{region " SIGNAL AREA : NAME->X_Pr_Axl3_Wh1 LENGTH->8 STARTBIT :0"}
Raw_X_Pr_Axl3_Wh1						:= _FB_CanRx_Message_224.X_Byte_0;
GVL.IIVD.X_Pr_Axl3_Wh1.e				:= (Raw_X_Pr_Axl3_Wh1 > 16#FD) AND (Raw_X_Pr_Axl3_Wh1 < 16#FF);
GVL.IIVD.X_Pr_Axl3_Wh1.na				:= (Raw_X_Pr_Axl3_Wh1 = 16#FF);
GVL.IIVD.X_Pr_Axl3_Wh1.RangeExcd		:= NOT ((USINT_TO_REAL(BYTE_TO_USINT(Raw_X_Pr_Axl3_Wh1)) >= 0) AND (USINT_TO_REAL(BYTE_TO_USINT(Raw_X_Pr_Axl3_Wh1)) <= 250));
GVL.IIVD.X_Pr_Axl3_Wh1.v				:= NOT( GVL.IIVD.S_TmOut_Lastik_Basinclari_2_0X224 OR GVL.IIVD.X_Pr_Axl3_Wh1.RangeExcd OR GVL.IIVD.X_Pr_Axl3_Wh1.e OR GVL.IIVD.X_Pr_Axl3_Wh1.na) ;
GVL.IIVD.X_Pr_Axl3_Wh1.x				:= 
(*SELECT 1 : Is data valid ?*)				SEL(GVL.IIVD.X_Pr_Axl3_Wh1.v,
(*DEFAULT value assigment*)					0,
(*Transmission is VALID*)					USINT_TO_REAL(BYTE_TO_USINT(Raw_X_Pr_Axl3_Wh1)));
{endregion}
{region " SIGNAL AREA : NAME->X_Pr_Axl3_Wh2 LENGTH->8 STARTBIT :8"}
Raw_X_Pr_Axl3_Wh2						:= _FB_CanRx_Message_224.X_Byte_1;
GVL.IIVD.X_Pr_Axl3_Wh2.e				:= (Raw_X_Pr_Axl3_Wh2 > 16#FD) AND (Raw_X_Pr_Axl3_Wh2 < 16#FF);
GVL.IIVD.X_Pr_Axl3_Wh2.na				:= (Raw_X_Pr_Axl3_Wh2 = 16#FF);
GVL.IIVD.X_Pr_Axl3_Wh2.RangeExcd		:= NOT ((USINT_TO_REAL(BYTE_TO_USINT(Raw_X_Pr_Axl3_Wh2)) >= 0) AND (USINT_TO_REAL(BYTE_TO_USINT(Raw_X_Pr_Axl3_Wh2)) <= 250));
GVL.IIVD.X_Pr_Axl3_Wh2.v				:= NOT( GVL.IIVD.S_TmOut_Lastik_Basinclari_2_0X224 OR GVL.IIVD.X_Pr_Axl3_Wh2.RangeExcd OR GVL.IIVD.X_Pr_Axl3_Wh2.e OR GVL.IIVD.X_Pr_Axl3_Wh2.na) ;
GVL.IIVD.X_Pr_Axl3_Wh2.x				:= 
(*SELECT 1 : Is data valid ?*)				SEL(GVL.IIVD.X_Pr_Axl3_Wh2.v,
(*DEFAULT value assigment*)					0,
(*Transmission is VALID*)					USINT_TO_REAL(BYTE_TO_USINT(Raw_X_Pr_Axl3_Wh2)));
{endregion}
{region " SIGNAL AREA : NAME->X_Pr_Axl3_Wh3 LENGTH->8 STARTBIT :16"}
Raw_X_Pr_Axl3_Wh3						:= _FB_CanRx_Message_224.X_Byte_2;
GVL.IIVD.X_Pr_Axl3_Wh3.e				:= (Raw_X_Pr_Axl3_Wh3 > 16#FD) AND (Raw_X_Pr_Axl3_Wh3 < 16#FF);
GVL.IIVD.X_Pr_Axl3_Wh3.na				:= (Raw_X_Pr_Axl3_Wh3 = 16#FF);
GVL.IIVD.X_Pr_Axl3_Wh3.RangeExcd		:= NOT ((USINT_TO_REAL(BYTE_TO_USINT(Raw_X_Pr_Axl3_Wh3)) >= 0) AND (USINT_TO_REAL(BYTE_TO_USINT(Raw_X_Pr_Axl3_Wh3)) <= 250));
GVL.IIVD.X_Pr_Axl3_Wh3.v				:= NOT( GVL.IIVD.S_TmOut_Lastik_Basinclari_2_0X224 OR GVL.IIVD.X_Pr_Axl3_Wh3.RangeExcd OR GVL.IIVD.X_Pr_Axl3_Wh3.e OR GVL.IIVD.X_Pr_Axl3_Wh3.na) ;
GVL.IIVD.X_Pr_Axl3_Wh3.x				:= 
(*SELECT 1 : Is data valid ?*)				SEL(GVL.IIVD.X_Pr_Axl3_Wh3.v,
(*DEFAULT value assigment*)					0,
(*Transmission is VALID*)					USINT_TO_REAL(BYTE_TO_USINT(Raw_X_Pr_Axl3_Wh3)));
{endregion}
{region " SIGNAL AREA : NAME->X_Pr_Axl3_Wh4 LENGTH->8 STARTBIT :24"}
Raw_X_Pr_Axl3_Wh4						:= _FB_CanRx_Message_224.X_Byte_3;
GVL.IIVD.X_Pr_Axl3_Wh4.e				:= (Raw_X_Pr_Axl3_Wh4 > 16#FD) AND (Raw_X_Pr_Axl3_Wh4 < 16#FF);
GVL.IIVD.X_Pr_Axl3_Wh4.na				:= (Raw_X_Pr_Axl3_Wh4 = 16#FF);
GVL.IIVD.X_Pr_Axl3_Wh4.RangeExcd		:= NOT ((USINT_TO_REAL(BYTE_TO_USINT(Raw_X_Pr_Axl3_Wh4)) >= 0) AND (USINT_TO_REAL(BYTE_TO_USINT(Raw_X_Pr_Axl3_Wh4)) <= 250));
GVL.IIVD.X_Pr_Axl3_Wh4.v				:= NOT( GVL.IIVD.S_TmOut_Lastik_Basinclari_2_0X224 OR GVL.IIVD.X_Pr_Axl3_Wh4.RangeExcd OR GVL.IIVD.X_Pr_Axl3_Wh4.e OR GVL.IIVD.X_Pr_Axl3_Wh4.na) ;
GVL.IIVD.X_Pr_Axl3_Wh4.x				:= 
(*SELECT 1 : Is data valid ?*)				SEL(GVL.IIVD.X_Pr_Axl3_Wh4.v,
(*DEFAULT value assigment*)					0,
(*Transmission is VALID*)					USINT_TO_REAL(BYTE_TO_USINT(Raw_X_Pr_Axl3_Wh4)));
{endregion}
{region " SIGNAL AREA : NAME->X_Pr_Axl4_Wh1 LENGTH->8 STARTBIT :32"}
Raw_X_Pr_Axl4_Wh1						:= _FB_CanRx_Message_224.X_Byte_4;
GVL.IIVD.X_Pr_Axl4_Wh1.e				:= (Raw_X_Pr_Axl4_Wh1 > 16#FD) AND (Raw_X_Pr_Axl4_Wh1 < 16#FF);
GVL.IIVD.X_Pr_Axl4_Wh1.na				:= (Raw_X_Pr_Axl4_Wh1 = 16#FF);
GVL.IIVD.X_Pr_Axl4_Wh1.RangeExcd		:= NOT ((USINT_TO_REAL(BYTE_TO_USINT(Raw_X_Pr_Axl4_Wh1)) >= 0) AND (USINT_TO_REAL(BYTE_TO_USINT(Raw_X_Pr_Axl4_Wh1)) <= 250));
GVL.IIVD.X_Pr_Axl4_Wh1.v				:= NOT( GVL.IIVD.S_TmOut_Lastik_Basinclari_2_0X224 OR GVL.IIVD.X_Pr_Axl4_Wh1.RangeExcd OR GVL.IIVD.X_Pr_Axl4_Wh1.e OR GVL.IIVD.X_Pr_Axl4_Wh1.na) ;
GVL.IIVD.X_Pr_Axl4_Wh1.x				:= 
(*SELECT 1 : Is data valid ?*)				SEL(GVL.IIVD.X_Pr_Axl4_Wh1.v,
(*DEFAULT value assigment*)					0,
(*Transmission is VALID*)					USINT_TO_REAL(BYTE_TO_USINT(Raw_X_Pr_Axl4_Wh1)));
{endregion}
{region " SIGNAL AREA : NAME->X_Pr_Axl4_Wh2 LENGTH->8 STARTBIT :40"}
Raw_X_Pr_Axl4_Wh2						:= _FB_CanRx_Message_224.X_Byte_5;
GVL.IIVD.X_Pr_Axl4_Wh2.e				:= (Raw_X_Pr_Axl4_Wh2 > 16#FD) AND (Raw_X_Pr_Axl4_Wh2 < 16#FF);
GVL.IIVD.X_Pr_Axl4_Wh2.na				:= (Raw_X_Pr_Axl4_Wh2 = 16#FF);
GVL.IIVD.X_Pr_Axl4_Wh2.RangeExcd		:= NOT ((USINT_TO_REAL(BYTE_TO_USINT(Raw_X_Pr_Axl4_Wh2)) >= 0) AND (USINT_TO_REAL(BYTE_TO_USINT(Raw_X_Pr_Axl4_Wh2)) <= 250));
GVL.IIVD.X_Pr_Axl4_Wh2.v				:= NOT( GVL.IIVD.S_TmOut_Lastik_Basinclari_2_0X224 OR GVL.IIVD.X_Pr_Axl4_Wh2.RangeExcd OR GVL.IIVD.X_Pr_Axl4_Wh2.e OR GVL.IIVD.X_Pr_Axl4_Wh2.na) ;
GVL.IIVD.X_Pr_Axl4_Wh2.x				:= 
(*SELECT 1 : Is data valid ?*)				SEL(GVL.IIVD.X_Pr_Axl4_Wh2.v,
(*DEFAULT value assigment*)					0,
(*Transmission is VALID*)					USINT_TO_REAL(BYTE_TO_USINT(Raw_X_Pr_Axl4_Wh2)));
{endregion}
{region " SIGNAL AREA : NAME->X_Pr_Axl4_Wh3 LENGTH->8 STARTBIT :48"}
Raw_X_Pr_Axl4_Wh3						:= _FB_CanRx_Message_224.X_Byte_6;
GVL.IIVD.X_Pr_Axl4_Wh3.e				:= (Raw_X_Pr_Axl4_Wh3 > 16#FD) AND (Raw_X_Pr_Axl4_Wh3 < 16#FF);
GVL.IIVD.X_Pr_Axl4_Wh3.na				:= (Raw_X_Pr_Axl4_Wh3 = 16#FF);
GVL.IIVD.X_Pr_Axl4_Wh3.RangeExcd		:= NOT ((USINT_TO_REAL(BYTE_TO_USINT(Raw_X_Pr_Axl4_Wh3)) >= 0) AND (USINT_TO_REAL(BYTE_TO_USINT(Raw_X_Pr_Axl4_Wh3)) <= 250));
GVL.IIVD.X_Pr_Axl4_Wh3.v				:= NOT( GVL.IIVD.S_TmOut_Lastik_Basinclari_2_0X224 OR GVL.IIVD.X_Pr_Axl4_Wh3.RangeExcd OR GVL.IIVD.X_Pr_Axl4_Wh3.e OR GVL.IIVD.X_Pr_Axl4_Wh3.na) ;
GVL.IIVD.X_Pr_Axl4_Wh3.x				:= 
(*SELECT 1 : Is data valid ?*)				SEL(GVL.IIVD.X_Pr_Axl4_Wh3.v,
(*DEFAULT value assigment*)					0,
(*Transmission is VALID*)					USINT_TO_REAL(BYTE_TO_USINT(Raw_X_Pr_Axl4_Wh3)));
{endregion}
{region " SIGNAL AREA : NAME->X_Pr_Axl4_Wh4 LENGTH->8 STARTBIT :56"}
Raw_X_Pr_Axl4_Wh4						:= _FB_CanRx_Message_224.X_Byte_7;
GVL.IIVD.X_Pr_Axl4_Wh4.e				:= (Raw_X_Pr_Axl4_Wh4 > 16#FD) AND (Raw_X_Pr_Axl4_Wh4 < 16#FF);
GVL.IIVD.X_Pr_Axl4_Wh4.na				:= (Raw_X_Pr_Axl4_Wh4 = 16#FF);
GVL.IIVD.X_Pr_Axl4_Wh4.RangeExcd		:= NOT ((USINT_TO_REAL(BYTE_TO_USINT(Raw_X_Pr_Axl4_Wh4)) >= 0) AND (USINT_TO_REAL(BYTE_TO_USINT(Raw_X_Pr_Axl4_Wh4)) <= 250));
GVL.IIVD.X_Pr_Axl4_Wh4.v				:= NOT( GVL.IIVD.S_TmOut_Lastik_Basinclari_2_0X224 OR GVL.IIVD.X_Pr_Axl4_Wh4.RangeExcd OR GVL.IIVD.X_Pr_Axl4_Wh4.e OR GVL.IIVD.X_Pr_Axl4_Wh4.na) ;
GVL.IIVD.X_Pr_Axl4_Wh4.x				:= 
(*SELECT 1 : Is data valid ?*)				SEL(GVL.IIVD.X_Pr_Axl4_Wh4.v,
(*DEFAULT value assigment*)					0,
(*Transmission is VALID*)					USINT_TO_REAL(BYTE_TO_USINT(Raw_X_Pr_Axl4_Wh4)));
{endregion}
{endregion}

{region " MESSAGE AREA :Arac_Bilgilendirme- ID:225"}

_FB_CanRx_Message_Unpack_225 (		C_Enable	:= GVL.IIVD.S_CAN_Init,
     								Obj_CAN		:= ADR(GVL.IC.Obj_CAN0),
     								X_MsgID		:= 16#225,
     								Tm_MsgTmOut	:= TIME#2500MS,
     								S_Extended	:= 0,
     								S_ER_TmOut	=> GVL.IIVD.S_TmOut_Arac_Bilgilendirme_0X225);

{region " SIGNAL AREA : NAME->S_Cvr_Op_Dr1_Ext LENGTH->2 STARTBIT :0"}
GVL.IIVD.S_Cvr_Op_Dr1_Ext.v				:= NOT GVL.IIVD.S_TmOut_Arac_Bilgilendirme_0X225 AND NOT _FB_CanRx_Message_Unpack_225.S_Bit_1;
GVL.IIVD.S_Cvr_Op_Dr1_Ext.x				:= GVL.IIVD.S_Cvr_Op_Dr1_Ext.v AND _FB_CanRx_Message_Unpack_225.S_Bit_0;
GVL.IIVD.S_Cvr_Op_Dr1_Ext.e				:= _FB_CanRx_Message_Unpack_225.S_Bit_1 AND NOT _FB_CanRx_Message_Unpack_225.S_Bit_0 ;
GVL.IIVD.S_Cvr_Op_Dr1_Ext.na			:= _FB_CanRx_Message_Unpack_225.S_Bit_1 AND _FB_CanRx_Message_Unpack_225.S_Bit_0 ;
{endregion}
{region " SIGNAL AREA : NAME->S_Cvr_Op_Lic LENGTH->2 STARTBIT :2"}
GVL.IIVD.S_Cvr_Op_Lic.v					:= NOT GVL.IIVD.S_TmOut_Arac_Bilgilendirme_0X225 AND NOT _FB_CanRx_Message_Unpack_225.S_Bit_3;
GVL.IIVD.S_Cvr_Op_Lic.x					:= GVL.IIVD.S_Cvr_Op_Lic.v AND _FB_CanRx_Message_Unpack_225.S_Bit_2;
GVL.IIVD.S_Cvr_Op_Lic.e					:= _FB_CanRx_Message_Unpack_225.S_Bit_3 AND NOT _FB_CanRx_Message_Unpack_225.S_Bit_2 ;
GVL.IIVD.S_Cvr_Op_Lic.na				:= _FB_CanRx_Message_Unpack_225.S_Bit_3 AND _FB_CanRx_Message_Unpack_225.S_Bit_2 ;
{endregion}
{region " SIGNAL AREA : NAME->S_Cvr_Op_Bat_Room LENGTH->2 STARTBIT :4"}
GVL.IIVD.S_Cvr_Op_Bat_Room.v			:= NOT GVL.IIVD.S_TmOut_Arac_Bilgilendirme_0X225 AND NOT _FB_CanRx_Message_Unpack_225.S_Bit_5;
GVL.IIVD.S_Cvr_Op_Bat_Room.x			:= GVL.IIVD.S_Cvr_Op_Bat_Room.v AND _FB_CanRx_Message_Unpack_225.S_Bit_4;
GVL.IIVD.S_Cvr_Op_Bat_Room.e			:= _FB_CanRx_Message_Unpack_225.S_Bit_5 AND NOT _FB_CanRx_Message_Unpack_225.S_Bit_4 ;
GVL.IIVD.S_Cvr_Op_Bat_Room.na			:= _FB_CanRx_Message_Unpack_225.S_Bit_5 AND _FB_CanRx_Message_Unpack_225.S_Bit_4 ;
{endregion}
{region " SIGNAL AREA : NAME->S_Cvr_Op_Mot LENGTH->2 STARTBIT :10"}
GVL.IIVD.S_Cvr_Op_Mot.v					:= NOT GVL.IIVD.S_TmOut_Arac_Bilgilendirme_0X225 AND NOT _FB_CanRx_Message_Unpack_225.S_Bit_11;
GVL.IIVD.S_Cvr_Op_Mot.x					:= GVL.IIVD.S_Cvr_Op_Mot.v AND _FB_CanRx_Message_Unpack_225.S_Bit_10;
GVL.IIVD.S_Cvr_Op_Mot.e					:= _FB_CanRx_Message_Unpack_225.S_Bit_11 AND NOT _FB_CanRx_Message_Unpack_225.S_Bit_10 ;
GVL.IIVD.S_Cvr_Op_Mot.na				:= _FB_CanRx_Message_Unpack_225.S_Bit_11 AND _FB_CanRx_Message_Unpack_225.S_Bit_10 ;
{endregion}
{region " SIGNAL AREA : NAME->S_Cvr_Op_Bwd_Lft_Chrg LENGTH->2 STARTBIT :12"}
GVL.IIVD.S_Cvr_Op_Bwd_Lft_Chrg.v		:= NOT GVL.IIVD.S_TmOut_Arac_Bilgilendirme_0X225 AND NOT _FB_CanRx_Message_Unpack_225.S_Bit_13;
GVL.IIVD.S_Cvr_Op_Bwd_Lft_Chrg.x		:= GVL.IIVD.S_Cvr_Op_Bwd_Lft_Chrg.v AND _FB_CanRx_Message_Unpack_225.S_Bit_12;
GVL.IIVD.S_Cvr_Op_Bwd_Lft_Chrg.e		:= _FB_CanRx_Message_Unpack_225.S_Bit_13 AND NOT _FB_CanRx_Message_Unpack_225.S_Bit_12 ;
GVL.IIVD.S_Cvr_Op_Bwd_Lft_Chrg.na		:= _FB_CanRx_Message_Unpack_225.S_Bit_13 AND _FB_CanRx_Message_Unpack_225.S_Bit_12 ;
{endregion}
{region " SIGNAL AREA : NAME->S_Cvr_Op_24V_Chrg_Plg LENGTH->2 STARTBIT :14"}
GVL.IIVD.S_Cvr_Op_24V_Chrg_Plg.v		:= NOT GVL.IIVD.S_TmOut_Arac_Bilgilendirme_0X225 AND NOT _FB_CanRx_Message_Unpack_225.S_Bit_15;
GVL.IIVD.S_Cvr_Op_24V_Chrg_Plg.x		:= GVL.IIVD.S_Cvr_Op_24V_Chrg_Plg.v AND _FB_CanRx_Message_Unpack_225.S_Bit_14;
GVL.IIVD.S_Cvr_Op_24V_Chrg_Plg.e		:= _FB_CanRx_Message_Unpack_225.S_Bit_15 AND NOT _FB_CanRx_Message_Unpack_225.S_Bit_14;
GVL.IIVD.S_Cvr_Op_24V_Chrg_Plg.na		:= _FB_CanRx_Message_Unpack_225.S_Bit_15 AND _FB_CanRx_Message_Unpack_225.S_Bit_14;
{endregion}
{region " SIGNAL AREA : NAME->S_Cvr_Op_Bwd LENGTH->2 STARTBIT :16"}
GVL.IIVD.S_Cvr_Op_Bwd.v					:= NOT GVL.IIVD.S_TmOut_Arac_Bilgilendirme_0X225 AND NOT _FB_CanRx_Message_Unpack_225.S_Bit_17;
GVL.IIVD.S_Cvr_Op_Bwd.x					:= GVL.IIVD.S_Cvr_Op_Bwd.v AND _FB_CanRx_Message_Unpack_225.S_Bit_16;
GVL.IIVD.S_Cvr_Op_Bwd.e					:= _FB_CanRx_Message_Unpack_225.S_Bit_17 AND NOT _FB_CanRx_Message_Unpack_225.S_Bit_16 ;
GVL.IIVD.S_Cvr_Op_Bwd.na				:= _FB_CanRx_Message_Unpack_225.S_Bit_17 AND _FB_CanRx_Message_Unpack_225.S_Bit_16 ;
{endregion}
{region " SIGNAL AREA : NAME->S_Rp_Op LENGTH->2 STARTBIT :18"}
GVL.IIVD.S_Rp_Op.v						:= NOT GVL.IIVD.S_TmOut_Arac_Bilgilendirme_0X225 AND NOT _FB_CanRx_Message_Unpack_225.S_Bit_19;
GVL.IIVD.S_Rp_Op.x						:= GVL.IIVD.S_Rp_Op.v AND _FB_CanRx_Message_Unpack_225.S_Bit_18;
GVL.IIVD.S_Rp_Op.e						:= _FB_CanRx_Message_Unpack_225.S_Bit_19 AND NOT _FB_CanRx_Message_Unpack_225.S_Bit_18 ;
GVL.IIVD.S_Rp_Op.na						:= _FB_CanRx_Message_Unpack_225.S_Bit_19 AND _FB_CanRx_Message_Unpack_225.S_Bit_18 ;
{endregion}
{region " SIGNAL AREA : NAME->S_Cvr_Op_Bwd_Mnt_Pnl LENGTH->2 STARTBIT :20"}
GVL.IIVD.S_Cvr_Op_Bwd_Mnt_Pnl.v			:= NOT GVL.IIVD.S_TmOut_Arac_Bilgilendirme_0X225 AND NOT _FB_CanRx_Message_Unpack_225.S_Bit_21;
GVL.IIVD.S_Cvr_Op_Bwd_Mnt_Pnl.x			:= GVL.IIVD.S_Cvr_Op_Bwd_Mnt_Pnl.v AND _FB_CanRx_Message_Unpack_225.S_Bit_20;
GVL.IIVD.S_Cvr_Op_Bwd_Mnt_Pnl.e			:= _FB_CanRx_Message_Unpack_225.S_Bit_21 AND NOT _FB_CanRx_Message_Unpack_225.S_Bit_20 ;
GVL.IIVD.S_Cvr_Op_Bwd_Mnt_Pnl.na		:= _FB_CanRx_Message_Unpack_225.S_Bit_21 AND _FB_CanRx_Message_Unpack_225.S_Bit_20 ;
{endregion}
{region " SIGNAL AREA : NAME->S_Cvr_Op_Bwd_Mnt_Pnl LENGTH->2 STARTBIT :22"}
GVL.IIVD.S_Cvr_Op_Frnt_Mnt_Pnl.v		:= NOT GVL.IIVD.S_TmOut_Arac_Bilgilendirme_0X225 AND NOT _FB_CanRx_Message_Unpack_225.S_Bit_23;
GVL.IIVD.S_Cvr_Op_Frnt_Mnt_Pnl.x		:= GVL.IIVD.S_Cvr_Op_Frnt_Mnt_Pnl.v AND _FB_CanRx_Message_Unpack_225.S_Bit_22;
GVL.IIVD.S_Cvr_Op_Frnt_Mnt_Pnl.e		:= _FB_CanRx_Message_Unpack_225.S_Bit_23 AND NOT _FB_CanRx_Message_Unpack_225.S_Bit_22 ;
GVL.IIVD.S_Cvr_Op_Frnt_Mnt_Pnl.na		:= _FB_CanRx_Message_Unpack_225.S_Bit_23 AND _FB_CanRx_Message_Unpack_225.S_Bit_22 ;
{endregion}
{region " SIGNAL AREA : NAME->S_ER_Rp_Op_Unauth LENGTH->2 STARTBIT :30"}
GVL.IIVD.S_ER_Rp_Op_Unauth.v			:= NOT GVL.IIVD.S_TmOut_Arac_Bilgilendirme_0X225 AND NOT _FB_CanRx_Message_Unpack_225.S_Bit_31;
GVL.IIVD.S_ER_Rp_Op_Unauth.x			:= GVL.IIVD.S_ER_Rp_Op_Unauth.v AND _FB_CanRx_Message_Unpack_225.S_Bit_30;
GVL.IIVD.S_ER_Rp_Op_Unauth.e			:= _FB_CanRx_Message_Unpack_225.S_Bit_31 AND NOT _FB_CanRx_Message_Unpack_225.S_Bit_30;
GVL.IIVD.S_ER_Rp_Op_Unauth.na			:= _FB_CanRx_Message_Unpack_225.S_Bit_31 AND _FB_CanRx_Message_Unpack_225.S_Bit_30;
{endregion}
{region " SIGNAL AREA : NAME->S_ER_Fi_Bat_Room LENGTH->2 STARTBIT :32"}
GVL.IIVD.S_ER_Fi_Bat_Room.v				:= NOT GVL.IIVD.S_TmOut_Arac_Bilgilendirme_0X225 AND NOT _FB_CanRx_Message_Unpack_225.S_Bit_33;
GVL.IIVD.S_ER_Fi_Bat_Room.x				:= GVL.IIVD.S_ER_Fi_Bat_Room.v AND _FB_CanRx_Message_Unpack_225.S_Bit_32;
GVL.IIVD.S_ER_Fi_Bat_Room.e				:= _FB_CanRx_Message_Unpack_225.S_Bit_33 AND NOT _FB_CanRx_Message_Unpack_225.S_Bit_32 ;
GVL.IIVD.S_ER_Fi_Bat_Room.na			:= _FB_CanRx_Message_Unpack_225.S_Bit_33 AND _FB_CanRx_Message_Unpack_225.S_Bit_32 ;
{endregion}
{region " SIGNAL AREA : NAME->S_ER_Not_Ins_Fi_Sens_Bat_Room LENGTH->2 STARTBIT :34"}
GVL.IIVD.S_ER_Not_Ins_Fi_Sens_Bat_Room.v	:= NOT GVL.IIVD.S_TmOut_Arac_Bilgilendirme_0X225 AND NOT _FB_CanRx_Message_Unpack_225.S_Bit_35;
GVL.IIVD.S_ER_Not_Ins_Fi_Sens_Bat_Room.x	:= GVL.IIVD.S_ER_Not_Ins_Fi_Sens_Bat_Room.v AND _FB_CanRx_Message_Unpack_225.S_Bit_34;
GVL.IIVD.S_ER_Not_Ins_Fi_Sens_Bat_Room.e	:= _FB_CanRx_Message_Unpack_225.S_Bit_35 AND NOT _FB_CanRx_Message_Unpack_225.S_Bit_34 ;
GVL.IIVD.S_ER_Not_Ins_Fi_Sens_Bat_Room.na	:= _FB_CanRx_Message_Unpack_225.S_Bit_35 AND _FB_CanRx_Message_Unpack_225.S_Bit_34 ;
{endregion}
{region " SIGNAL AREA : NAME->S_ER_Fi_Frnt_Pnl LENGTH->2 STARTBIT :36"}
GVL.IIVD.S_ER_Fi_Frnt_Pnl.v				:= NOT GVL.IIVD.S_TmOut_Arac_Bilgilendirme_0X225 AND NOT _FB_CanRx_Message_Unpack_225.S_Bit_37;
GVL.IIVD.S_ER_Fi_Frnt_Pnl.x				:= GVL.IIVD.S_ER_Fi_Frnt_Pnl.v AND _FB_CanRx_Message_Unpack_225.S_Bit_36;
GVL.IIVD.S_ER_Fi_Frnt_Pnl.e				:= _FB_CanRx_Message_Unpack_225.S_Bit_37 AND NOT _FB_CanRx_Message_Unpack_225.S_Bit_36 ;
GVL.IIVD.S_ER_Fi_Frnt_Pnl.na			:= _FB_CanRx_Message_Unpack_225.S_Bit_37 AND _FB_CanRx_Message_Unpack_225.S_Bit_36 ;
{endregion}
{region " SIGNAL AREA : NAME->S_ER_Not_Ins_Fi_Snsr_Frnt_Pnl LENGTH->2 STARTBIT :38"}
GVL.IIVD.S_ER_Not_Ins_Fi_Snsr_Frnt_Pnl.v	:= NOT GVL.IIVD.S_TmOut_Arac_Bilgilendirme_0X225 AND NOT _FB_CanRx_Message_Unpack_225.S_Bit_39;
GVL.IIVD.S_ER_Not_Ins_Fi_Snsr_Frnt_Pnl.x	:= GVL.IIVD.S_ER_Not_Ins_Fi_Snsr_Frnt_Pnl.v AND _FB_CanRx_Message_Unpack_225.S_Bit_38;
GVL.IIVD.S_ER_Not_Ins_Fi_Snsr_Frnt_Pnl.e	:= _FB_CanRx_Message_Unpack_225.S_Bit_39 AND NOT _FB_CanRx_Message_Unpack_225.S_Bit_38 ;
GVL.IIVD.S_ER_Not_Ins_Fi_Snsr_Frnt_Pnl.na	:= _FB_CanRx_Message_Unpack_225.S_Bit_39 AND _FB_CanRx_Message_Unpack_225.S_Bit_38 ;
{endregion}
{region " SIGNAL AREA : NAME->S_ER_Fi_Drv_Mot LENGTH->2 STARTBIT :40"}
GVL.IIVD.S_ER_Fi_Drv_Mot.v				:= NOT GVL.IIVD.S_TmOut_Arac_Bilgilendirme_0X225 AND NOT _FB_CanRx_Message_Unpack_225.S_Bit_41;
GVL.IIVD.S_ER_Fi_Drv_Mot.x				:= GVL.IIVD.S_ER_Fi_Drv_Mot.v AND _FB_CanRx_Message_Unpack_225.S_Bit_40;
GVL.IIVD.S_ER_Fi_Drv_Mot.e				:= _FB_CanRx_Message_Unpack_225.S_Bit_41 AND NOT _FB_CanRx_Message_Unpack_225.S_Bit_40 ;
GVL.IIVD.S_ER_Fi_Drv_Mot.na				:= _FB_CanRx_Message_Unpack_225.S_Bit_41 AND _FB_CanRx_Message_Unpack_225.S_Bit_40 ;
{endregion}
{region " SIGNAL AREA : NAME->S_ER_Not_Ins_Fi_Snsr_Drv_Mot LENGTH->2 STARTBIT :42"}
GVL.IIVD.S_ER_Not_Ins_Fi_Snsr_Drv_Mot.v		:= NOT GVL.IIVD.S_TmOut_Arac_Bilgilendirme_0X225 AND NOT _FB_CanRx_Message_Unpack_225.S_Bit_43;
GVL.IIVD.S_ER_Not_Ins_Fi_Snsr_Drv_Mot.x		:= GVL.IIVD.S_ER_Not_Ins_Fi_Snsr_Drv_Mot.v AND _FB_CanRx_Message_Unpack_225.S_Bit_42;
GVL.IIVD.S_ER_Not_Ins_Fi_Snsr_Drv_Mot.e		:= _FB_CanRx_Message_Unpack_225.S_Bit_43 AND NOT _FB_CanRx_Message_Unpack_225.S_Bit_42 ;
GVL.IIVD.S_ER_Not_Ins_Fi_Snsr_Drv_Mot.na	:= _FB_CanRx_Message_Unpack_225.S_Bit_43 AND _FB_CanRx_Message_Unpack_225.S_Bit_42 ;
{endregion}
{region " SIGNAL AREA : NAME->S_ER_Fi_Bwd_Pnl LENGTH->2 STARTBIT :44"}
GVL.IIVD.S_ER_Fi_Bwd_Pnl.v					:= NOT GVL.IIVD.S_TmOut_Arac_Bilgilendirme_0X225 AND NOT _FB_CanRx_Message_Unpack_225.S_Bit_45;
GVL.IIVD.S_ER_Fi_Bwd_Pnl.x					:= GVL.IIVD.S_ER_Fi_Bwd_Pnl.v AND _FB_CanRx_Message_Unpack_225.S_Bit_44;
GVL.IIVD.S_ER_Fi_Bwd_Pnl.e					:= _FB_CanRx_Message_Unpack_225.S_Bit_45 AND NOT _FB_CanRx_Message_Unpack_225.S_Bit_44 ;
GVL.IIVD.S_ER_Fi_Bwd_Pnl.na					:= _FB_CanRx_Message_Unpack_225.S_Bit_45 AND _FB_CanRx_Message_Unpack_225.S_Bit_44 ;
{endregion}
{region " SIGNAL AREA : NAME->S_ER_Not_Ins_Fi_Snsr_Bwd_Pnl LENGTH->2 STARTBIT :46"}
GVL.IIVD.S_ER_Not_Ins_Fi_Snsr_Bwd_Pnl.v		:= NOT GVL.IIVD.S_TmOut_Arac_Bilgilendirme_0X225 AND NOT _FB_CanRx_Message_Unpack_225.S_Bit_47;
GVL.IIVD.S_ER_Not_Ins_Fi_Snsr_Bwd_Pnl.x		:= GVL.IIVD.S_ER_Not_Ins_Fi_Snsr_Bwd_Pnl.v AND _FB_CanRx_Message_Unpack_225.S_Bit_46;
GVL.IIVD.S_ER_Not_Ins_Fi_Snsr_Bwd_Pnl.e		:= _FB_CanRx_Message_Unpack_225.S_Bit_47 AND NOT _FB_CanRx_Message_Unpack_225.S_Bit_46 ;
GVL.IIVD.S_ER_Not_Ins_Fi_Snsr_Bwd_Pnl.na	:= _FB_CanRx_Message_Unpack_225.S_Bit_47 AND _FB_CanRx_Message_Unpack_225.S_Bit_46 ;
{endregion}
{region " SIGNAL AREA : NAME->S_ER_Fi_Eng_Room LENGTH->2 STARTBIT :48"}
GVL.IIVD.S_ER_Fi_Eng_Room.v					:= NOT GVL.IIVD.S_TmOut_Arac_Bilgilendirme_0X225 AND NOT _FB_CanRx_Message_Unpack_225.S_Bit_49;
GVL.IIVD.S_ER_Fi_Eng_Room.x					:= GVL.IIVD.S_ER_Fi_Eng_Room.v AND _FB_CanRx_Message_Unpack_225.S_Bit_48;
GVL.IIVD.S_ER_Fi_Eng_Room.e					:= _FB_CanRx_Message_Unpack_225.S_Bit_49 AND NOT _FB_CanRx_Message_Unpack_225.S_Bit_48 ;
GVL.IIVD.S_ER_Fi_Eng_Room.na				:= _FB_CanRx_Message_Unpack_225.S_Bit_49 AND _FB_CanRx_Message_Unpack_225.S_Bit_48 ;
{endregion}
{region " SIGNAL AREA : NAME->S_ER_Not_Ins_Fi_Sns_Eng_Room LENGTH->2 STARTBIT :50"}
GVL.IIVD.S_ER_Not_Ins_Fi_Sns_Eng_Room.v		:= NOT GVL.IIVD.S_TmOut_Arac_Bilgilendirme_0X225 AND NOT _FB_CanRx_Message_Unpack_225.S_Bit_51;
GVL.IIVD.S_ER_Not_Ins_Fi_Sns_Eng_Room.x		:= GVL.IIVD.S_ER_Not_Ins_Fi_Sns_Eng_Room.v AND _FB_CanRx_Message_Unpack_225.S_Bit_50;
GVL.IIVD.S_ER_Not_Ins_Fi_Sns_Eng_Room.e		:= _FB_CanRx_Message_Unpack_225.S_Bit_51 AND NOT _FB_CanRx_Message_Unpack_225.S_Bit_50 ;
GVL.IIVD.S_ER_Not_Ins_Fi_Sns_Eng_Room.na	:= _FB_CanRx_Message_Unpack_225.S_Bit_51 AND _FB_CanRx_Message_Unpack_225.S_Bit_50 ;
{endregion}
{endregion}

{region " MESSAGE AREA :Arac_Kritik_Uyarilari- ID:226"}

_FB_CanRx_Message_Unpack_226 (	C_Enable	:= GVL.IIVD.S_CAN_Init,
     							Obj_CAN		:= ADR(GVL.IC.Obj_CAN0),
     							X_MsgID		:= 16#226,
     							Tm_MsgTmOut	:= TIME#2500MS,
     							S_Extended	:= 0,
     							S_ER_TmOut	=> GVL.IIVD.S_TmOut_Arac_Kritik_Uyarilari_0X226);

{region " SIGNAL AREA : NAME->X_Psng_No LENGTH->8 STARTBIT :0"}
Raw_X_Psng_No							:= _FB_CanRx_Message_Unpack_226.X_Byte_0;
GVL.IIVD.X_Psng_No.e					:= (Raw_X_Psng_No > 16#FD) AND (Raw_X_Psng_No < 16#FF);
GVL.IIVD.X_Psng_No.na					:= (Raw_X_Psng_No = 16#FF);
GVL.IIVD.X_Psng_No.RangeExcd			:= NOT ((USINT_TO_REAL(BYTE_TO_USINT(Raw_X_Psng_No)) >= 0) AND (USINT_TO_REAL(BYTE_TO_USINT(Raw_X_Psng_No)) <= 250));
GVL.IIVD.X_Psng_No.v					:= NOT( GVL.IIVD.S_TmOut_Arac_Kritik_Uyarilari_0X226 OR GVL.IIVD.X_Psng_No.RangeExcd OR GVL.IIVD.X_Psng_No.e OR GVL.IIVD.X_Psng_No.na) ;
GVL.IIVD.X_Psng_No.x					:= 
(*SELECT 1 : Is data valid ?*)				SEL(GVL.IIVD.X_Psng_No.v,
(*DEFAULT value assigment*)					0,
(*Transmission is VALID*)					USINT_TO_REAL(BYTE_TO_USINT(Raw_X_Psng_No)));
{endregion}
{region " SIGNAL AREA : NAME->X_Wgt_Axle LENGTH->16 STARTBIT :8"}
_FB_PACK_BYTE_TO_WORD_4 (	X_BYTE_0	:= _FB_CanRx_Message_Unpack_226.X_Byte_1, 
							X_BYTE_1	:= _FB_CanRx_Message_Unpack_226.X_Byte_2, 
							X_WORD_0 	=> Raw_X_Wgt_Axle);
GVL.IIVD.X_Wgt_Axle.e					:= (Raw_X_Wgt_Axle > 16#FDFF) AND (Raw_X_Wgt_Axle <= 16#FEFF);
GVL.IIVD.X_Wgt_Axle.na					:= (Raw_X_Wgt_Axle > 16#FEFF);
GVL.IIVD.X_Wgt_Axle.RangeExcd			:= NOT ((UINT_TO_REAL(WORD_TO_UINT(Raw_X_Wgt_Axle)) >= 0) AND (UINT_TO_REAL(WORD_TO_UINT(Raw_X_Wgt_Axle)) <= 65000));
GVL.IIVD.X_Wgt_Axle.v					:= NOT( GVL.IIVD.S_TmOut_Arac_Kritik_Uyarilari_0X226 OR GVL.IIVD.X_Wgt_Axle.RangeExcd OR GVL.IIVD.X_Wgt_Axle.e OR GVL.IIVD.X_Wgt_Axle.na) ;
GVL.IIVD.X_Wgt_Axle.x					:= 
(*SELECT 1 : Is data valid ?*)				SEL(GVL.IIVD.X_Wgt_Axle.v,
(*DEFAULT value assigment*)					0,
(*Transmission is VALID*)					UINT_TO_REAL(WORD_TO_UINT(Raw_X_Wgt_Axle)));
{endregion}
{region " SIGNAL AREA : NAME->C_Err_Pg_Dn LENGTH->2 STARTBIT :24"}
GVL.IIVD.C_Err_Pg_Dn.v					:= NOT GVL.IIVD.S_TmOut_Arac_Kritik_Uyarilari_0X226 AND NOT _FB_CanRx_Message_Unpack_226.S_Bit_25;
GVL.IIVD.C_Err_Pg_Dn.x					:= GVL.IIVD.C_Err_Pg_Dn.v AND _FB_CanRx_Message_Unpack_226.S_Bit_24;
GVL.IIVD.C_Err_Pg_Dn.e					:= _FB_CanRx_Message_Unpack_226.S_Bit_25 AND NOT _FB_CanRx_Message_Unpack_226.S_Bit_24 ;
GVL.IIVD.C_Err_Pg_Dn.na					:= _FB_CanRx_Message_Unpack_226.S_Bit_25 AND _FB_CanRx_Message_Unpack_226.S_Bit_24 ;
{endregion}
{region " SIGNAL AREA : NAME->C_Err_Pg_Up LENGTH->2 STARTBIT :26"}
GVL.IIVD.C_Err_Pg_Up.v					:= NOT GVL.IIVD.S_TmOut_Arac_Kritik_Uyarilari_0X226 AND NOT _FB_CanRx_Message_Unpack_226.S_Bit_27;
GVL.IIVD.C_Err_Pg_Up.x					:= GVL.IIVD.C_Err_Pg_Up.v AND _FB_CanRx_Message_Unpack_226.S_Bit_26;
GVL.IIVD.C_Err_Pg_Up.e					:= _FB_CanRx_Message_Unpack_226.S_Bit_27 AND NOT _FB_CanRx_Message_Unpack_226.S_Bit_26 ;
GVL.IIVD.C_Err_Pg_Up.na					:= _FB_CanRx_Message_Unpack_226.S_Bit_27 AND _FB_CanRx_Message_Unpack_226.S_Bit_26 ;
{endregion}
{region " SIGNAL AREA : NAME->C_Rst_Trip LENGTH->2 STARTBIT :28"}
GVL.IIVD.C_Rst_Trip.v					:= NOT GVL.IIVD.S_TmOut_Arac_Kritik_Uyarilari_0X226 AND NOT _FB_CanRx_Message_Unpack_226.S_Bit_29;
GVL.IIVD.C_Rst_Trip.x					:= GVL.IIVD.C_Rst_Trip.v AND _FB_CanRx_Message_Unpack_226.S_Bit_28;
GVL.IIVD.C_Rst_Trip.e					:= _FB_CanRx_Message_Unpack_226.S_Bit_29 AND NOT _FB_CanRx_Message_Unpack_226.S_Bit_28 ;
GVL.IIVD.C_Rst_Trip.na					:= _FB_CanRx_Message_Unpack_226.S_Bit_29 AND _FB_CanRx_Message_Unpack_226.S_Bit_28 ;
{endregion}								 
{region " SIGNAL AREA : NAME->S_Drug_Alch_Ctrl LENGTH->2 STARTBIT :32"}
GVL.IIVD.S_Drug_Alch_Ctrl.v				:= NOT GVL.IIVD.S_TmOut_Arac_Kritik_Uyarilari_0X226 AND NOT _FB_CanRx_Message_Unpack_226.S_Bit_33;
GVL.IIVD.S_Drug_Alch_Ctrl.x				:= GVL.IIVD.S_Drug_Alch_Ctrl.v AND _FB_CanRx_Message_Unpack_226.S_Bit_32;
GVL.IIVD.S_Drug_Alch_Ctrl.e				:= _FB_CanRx_Message_Unpack_226.S_Bit_33 AND NOT _FB_CanRx_Message_Unpack_226.S_Bit_32 ;
GVL.IIVD.S_Drug_Alch_Ctrl.na			:= _FB_CanRx_Message_Unpack_226.S_Bit_33 AND _FB_CanRx_Message_Unpack_226.S_Bit_32 ;
{endregion}
{region " SIGNAL AREA : NAME->S_Drug_Alch_Warn LENGTH->2 STARTBIT :34"}
GVL.IIVD.S_Drug_Alch_Warn.v				:= NOT GVL.IIVD.S_TmOut_Arac_Kritik_Uyarilari_0X226 AND NOT _FB_CanRx_Message_Unpack_226.S_Bit_35;
GVL.IIVD.S_Drug_Alch_Warn.x				:= GVL.IIVD.S_Drug_Alch_Warn.v AND _FB_CanRx_Message_Unpack_226.S_Bit_34;
GVL.IIVD.S_Drug_Alch_Warn.e				:= _FB_CanRx_Message_Unpack_226.S_Bit_35 AND NOT _FB_CanRx_Message_Unpack_226.S_Bit_34 ;
GVL.IIVD.S_Drug_Alch_Warn.na			:= _FB_CanRx_Message_Unpack_226.S_Bit_35 AND _FB_CanRx_Message_Unpack_226.S_Bit_34 ;
{endregion}  
// PR1006_REV_002729_TIMTRO
{region " SIGNAL AREA : NAME->C_Flr_Heat_Off LENGTH->2 STARTBIT :36"}
GVL.IIVD.S_Prheat_Tk_Lv_Lo.v			:= NOT GVL.IIVD.S_TmOut_Arac_Kritik_Uyarilari_0X226 AND NOT _FB_CanRx_Message_Unpack_226.S_Bit_37;
GVL.IIVD.S_Prheat_Tk_Lv_Lo.x			:= GVL.IIVD.S_Prheat_Tk_Lv_Lo.v AND _FB_CanRx_Message_Unpack_226.S_Bit_36;
GVL.IIVD.S_Prheat_Tk_Lv_Lo.e			:= _FB_CanRx_Message_Unpack_226.S_Bit_37 AND NOT _FB_CanRx_Message_Unpack_226.S_Bit_36 ;
GVL.IIVD.S_Prheat_Tk_Lv_Lo.na			:= _FB_CanRx_Message_Unpack_226.S_Bit_37 AND _FB_CanRx_Message_Unpack_226.S_Bit_36 ;
{endregion}		  				 
{region " SIGNAL AREA : NAME->S_ER_Wpr_Wtr_Lv LENGTH->2 STARTBIT :40"}
GVL.IIVD.S_ER_Wpr_Wtr_Lv.v				:= NOT GVL.IIVD.S_TmOut_Arac_Kritik_Uyarilari_0X226 AND NOT _FB_CanRx_Message_Unpack_226.S_Bit_41;
GVL.IIVD.S_ER_Wpr_Wtr_Lv.x				:= GVL.IIVD.S_ER_Wpr_Wtr_Lv.v AND _FB_CanRx_Message_Unpack_226.S_Bit_40;
GVL.IIVD.S_ER_Wpr_Wtr_Lv.e				:= _FB_CanRx_Message_Unpack_226.S_Bit_41 AND NOT _FB_CanRx_Message_Unpack_226.S_Bit_40 ;
GVL.IIVD.S_ER_Wpr_Wtr_Lv.na				:= _FB_CanRx_Message_Unpack_226.S_Bit_41 AND _FB_CanRx_Message_Unpack_226.S_Bit_40 ;
{endregion}
{region " SIGNAL AREA : NAME->S_Sfty_Belt_Ins LENGTH->2 STARTBIT :42"}
GVL.IIVD.S_Sfty_Belt_Ins.v				:= NOT GVL.IIVD.S_TmOut_Arac_Kritik_Uyarilari_0X226 AND NOT _FB_CanRx_Message_Unpack_226.S_Bit_43;
GVL.IIVD.S_Sfty_Belt_Ins.x				:= GVL.IIVD.S_Sfty_Belt_Ins.v AND _FB_CanRx_Message_Unpack_226.S_Bit_42;
GVL.IIVD.S_Sfty_Belt_Ins.e				:= _FB_CanRx_Message_Unpack_226.S_Bit_43 AND NOT _FB_CanRx_Message_Unpack_226.S_Bit_42 ;
GVL.IIVD.S_Sfty_Belt_Ins.na				:= _FB_CanRx_Message_Unpack_226.S_Bit_43 AND _FB_CanRx_Message_Unpack_226.S_Bit_42 ;
{endregion}  
{region " SIGNAL AREA : NAME->C_Pnt_Up LENGTH->2 STARTBIT :44"}
GVL.IIVD.C_Pnt_Up.v						:= NOT GVL.IIVD.S_TmOut_Arac_Kritik_Uyarilari_0X226 AND NOT _FB_CanRx_Message_Unpack_226.S_Bit_45;
GVL.IIVD.C_Pnt_Up.x						:= GVL.IIVD.C_Pnt_Up.v AND _FB_CanRx_Message_Unpack_226.S_Bit_44;
GVL.IIVD.C_Pnt_Up.e						:= _FB_CanRx_Message_Unpack_226.S_Bit_45 AND NOT _FB_CanRx_Message_Unpack_226.S_Bit_44 ;
GVL.IIVD.C_Pnt_Up.na					:= _FB_CanRx_Message_Unpack_226.S_Bit_45 AND _FB_CanRx_Message_Unpack_226.S_Bit_44 ;
{endregion}	
{region " SIGNAL AREA : NAME->C_Pnt_Dn LENGTH->2 STARTBIT :46"}
GVL.IIVD.C_Pnt_Dn.v						:= NOT GVL.IIVD.S_TmOut_Arac_Kritik_Uyarilari_0X226 AND NOT _FB_CanRx_Message_Unpack_226.S_Bit_47;
GVL.IIVD.C_Pnt_Dn.x						:= GVL.IIVD.C_Pnt_Dn.v AND _FB_CanRx_Message_Unpack_226.S_Bit_46;
GVL.IIVD.C_Pnt_Dn.e						:= _FB_CanRx_Message_Unpack_226.S_Bit_47 AND NOT _FB_CanRx_Message_Unpack_226.S_Bit_46 ;
GVL.IIVD.C_Pnt_Dn.na					:= _FB_CanRx_Message_Unpack_226.S_Bit_47 AND _FB_CanRx_Message_Unpack_226.S_Bit_46 ;
{endregion}			  
{region " SIGNAL AREA : NAME->S_Drv_Seat_Pre_Snsr LENGTH->2 STARTBIT :48"}
GVL.IIVD.S_Drv_Seat_Pre_Snsr.v			:= NOT GVL.IIVD.S_TmOut_Arac_Kritik_Uyarilari_0X226 AND NOT _FB_CanRx_Message_Unpack_226.S_Bit_49;
GVL.IIVD.S_Drv_Seat_Pre_Snsr.x			:= GVL.IIVD.S_Drv_Seat_Pre_Snsr.v AND _FB_CanRx_Message_Unpack_226.S_Bit_48;
GVL.IIVD.S_Drv_Seat_Pre_Snsr.e			:= _FB_CanRx_Message_Unpack_226.S_Bit_49 AND NOT _FB_CanRx_Message_Unpack_226.S_Bit_48;
GVL.IIVD.S_Drv_Seat_Pre_Snsr.na			:= _FB_CanRx_Message_Unpack_226.S_Bit_49 AND _FB_CanRx_Message_Unpack_226.S_Bit_48;
{endregion}	
{region " SIGNAL AREA : NAME->S_Inc_Acc LENGTH->2 STARTBIT :56"}
GVL.IIVD.S_Inc_Acc.v						:= NOT GVL.IIVD.S_TmOut_Arac_Kritik_Uyarilari_0X226 AND NOT _FB_CanRx_Message_Unpack_226.S_Bit_57;
GVL.IIVD.S_Inc_Acc.x						:= GVL.IIVD.S_Inc_Acc.v AND _FB_CanRx_Message_Unpack_226.S_Bit_56;
GVL.IIVD.S_Inc_Acc.e						:= _FB_CanRx_Message_Unpack_226.S_Bit_57 AND NOT _FB_CanRx_Message_Unpack_226.S_Bit_56;
GVL.IIVD.S_Inc_Acc.na						:= _FB_CanRx_Message_Unpack_226.S_Bit_57 AND _FB_CanRx_Message_Unpack_226.S_Bit_56;
{endregion}
{region " SIGNAL AREA : NAME->S_Inc_Stop LENGTH->2 STARTBIT :58"}
GVL.IIVD.S_Inc_Stop.v						:= NOT GVL.IIVD.S_TmOut_Arac_Kritik_Uyarilari_0X226 AND NOT _FB_CanRx_Message_Unpack_226.S_Bit_59;
GVL.IIVD.S_Inc_Stop.x						:= GVL.IIVD.S_Inc_Stop.v AND _FB_CanRx_Message_Unpack_226.S_Bit_58;
GVL.IIVD.S_Inc_Stop.e						:= _FB_CanRx_Message_Unpack_226.S_Bit_59 AND NOT _FB_CanRx_Message_Unpack_226.S_Bit_58;
GVL.IIVD.S_Inc_Stop.na						:= _FB_CanRx_Message_Unpack_226.S_Bit_59 AND _FB_CanRx_Message_Unpack_226.S_Bit_58;
{endregion}
{region " SIGNAL AREA : NAME->S_Er_Tire_Pres LENGTH->2 STARTBIT :60"}
GVL.IIVD.S_Er_Tire_Pres.v					:= NOT GVL.IIVD.S_TmOut_Arac_Kritik_Uyarilari_0X226 AND NOT _FB_CanRx_Message_Unpack_226.S_Bit_61;
GVL.IIVD.S_Er_Tire_Pres.x					:= GVL.IIVD.S_Er_Tire_Pres.v AND _FB_CanRx_Message_Unpack_226.S_Bit_60;
GVL.IIVD.S_Er_Tire_Pres.e					:= _FB_CanRx_Message_Unpack_226.S_Bit_61 AND NOT _FB_CanRx_Message_Unpack_226.S_Bit_60;
GVL.IIVD.S_Er_Tire_Pres.na					:= _FB_CanRx_Message_Unpack_226.S_Bit_61 AND _FB_CanRx_Message_Unpack_226.S_Bit_60;
{endregion}
{endregion}

{region " MESSAGE AREA :Kapi_Hatalari_1- ID:230"}

_FB_CanRx_Message_230 (		C_Enable	:= GVL.IIVD.S_CAN_Init,
     						Obj_CAN		:= ADR(GVL.IC.Obj_CAN0),
     						X_MsgID		:= 16#230,
     						Tm_MsgTmOut	:= TIME#2500MS,
     						S_Extended	:= 0,
     						S_ER_TmOut	=> GVL.IIVD.S_TmOut_Kapi_Hatalari_1_0X230);

{region " SIGNAL AREA : NAME->Z_Dr1_Err_Fram_1 LENGTH->8 STARTBIT :0"}
Raw_Z_Dr1_Err_Fram_1					:= _FB_CanRx_Message_230.X_Byte_0;
GVL.IIVD.Z_Dr1_Err_Fram_1.e				:= (Raw_Z_Dr1_Err_Fram_1 > 16#FD) AND (Raw_Z_Dr1_Err_Fram_1 < 16#FF);
GVL.IIVD.Z_Dr1_Err_Fram_1.na			:= (Raw_Z_Dr1_Err_Fram_1 = 16#FF);
GVL.IIVD.Z_Dr1_Err_Fram_1.RangeExcd		:= NOT ((Raw_Z_Dr1_Err_Fram_1 >= 0) AND (Raw_Z_Dr1_Err_Fram_1 <= 255));
GVL.IIVD.Z_Dr1_Err_Fram_1.v				:= NOT( GVL.IIVD.S_TmOut_Kapi_Hatalari_1_0X230 OR GVL.IIVD.Z_Dr1_Err_Fram_1.RangeExcd OR GVL.IIVD.Z_Dr1_Err_Fram_1.e OR GVL.IIVD.Z_Dr1_Err_Fram_1.na) ;
GVL.IIVD.Z_Dr1_Err_Fram_1.x				:= 
(*SELECT 1 : Is data valid ?*)				SEL(GVL.IIVD.Z_Dr1_Err_Fram_1.v,
(*DEFAULT value assigment*)					0,
(*Transmission is VALID*)					Raw_Z_Dr1_Err_Fram_1);
{endregion}
{region " SIGNAL AREA : NAME->Z_Dr1_Err_Fram_2 LENGTH->8 STARTBIT :8"}
Raw_Z_Dr1_Err_Fram_2					:= _FB_CanRx_Message_230.X_Byte_1;
GVL.IIVD.Z_Dr1_Err_Fram_2.e				:= (Raw_Z_Dr1_Err_Fram_2 > 16#FD) AND (Raw_Z_Dr1_Err_Fram_2 < 16#FF);
GVL.IIVD.Z_Dr1_Err_Fram_2.na			:= (Raw_Z_Dr1_Err_Fram_2 = 16#FF);
GVL.IIVD.Z_Dr1_Err_Fram_2.RangeExcd		:= NOT ((Raw_Z_Dr1_Err_Fram_2 >= 0) AND (Raw_Z_Dr1_Err_Fram_2 <= 255));
GVL.IIVD.Z_Dr1_Err_Fram_2.v				:= NOT( GVL.IIVD.S_TmOut_Kapi_Hatalari_1_0X230 OR GVL.IIVD.Z_Dr1_Err_Fram_2.RangeExcd OR GVL.IIVD.Z_Dr1_Err_Fram_2.e OR GVL.IIVD.Z_Dr1_Err_Fram_2.na) ;
GVL.IIVD.Z_Dr1_Err_Fram_2.x				:= 
(*SELECT 1 : Is data valid ?*)				SEL(GVL.IIVD.Z_Dr1_Err_Fram_2.v,
(*DEFAULT value assigment*)					0,
(*Transmission is VALID*)					Raw_Z_Dr1_Err_Fram_2);
{endregion}
{region " SIGNAL AREA : NAME->Z_Dr1_Err_Fram_3 LENGTH->8 STARTBIT :16"}
Raw_Z_Dr1_Err_Fram_3					:= _FB_CanRx_Message_230.X_Byte_2;
GVL.IIVD.Z_Dr1_Err_Fram_3.e				:= (Raw_Z_Dr1_Err_Fram_3 > 16#FD) AND (Raw_Z_Dr1_Err_Fram_3 < 16#FF);
GVL.IIVD.Z_Dr1_Err_Fram_3.na			:= (Raw_Z_Dr1_Err_Fram_3 = 16#FF);
GVL.IIVD.Z_Dr1_Err_Fram_3.RangeExcd		:= NOT ((Raw_Z_Dr1_Err_Fram_3 >= 0) AND (Raw_Z_Dr1_Err_Fram_3 <= 255));
GVL.IIVD.Z_Dr1_Err_Fram_3.v				:= NOT( GVL.IIVD.S_TmOut_Kapi_Hatalari_1_0X230 OR GVL.IIVD.Z_Dr1_Err_Fram_3.RangeExcd OR GVL.IIVD.Z_Dr1_Err_Fram_3.e OR GVL.IIVD.Z_Dr1_Err_Fram_3.na) ;
GVL.IIVD.Z_Dr1_Err_Fram_3.x				:= 
(*SELECT 1 : Is data valid ?*)				SEL(GVL.IIVD.Z_Dr1_Err_Fram_3.v,
(*DEFAULT value assigment*)					0,
(*Transmission is VALID*)					Raw_Z_Dr1_Err_Fram_3);
{endregion}
{region " SIGNAL AREA : NAME->Z_Dr2_Err_Fram_1 LENGTH->8 STARTBIT :32"}
Raw_Z_Dr2_Err_Fram_1					:= _FB_CanRx_Message_230.X_Byte_4;
GVL.IIVD.Z_Dr2_Err_Fram_1.e				:= (Raw_Z_Dr2_Err_Fram_1 > 16#FD) AND (Raw_Z_Dr2_Err_Fram_1 < 16#FF);
GVL.IIVD.Z_Dr2_Err_Fram_1.na			:= (Raw_Z_Dr2_Err_Fram_1 = 16#FF);
GVL.IIVD.Z_Dr2_Err_Fram_1.RangeExcd		:= NOT ((Raw_Z_Dr2_Err_Fram_1 >= 0) AND (Raw_Z_Dr2_Err_Fram_1 <= 255));
GVL.IIVD.Z_Dr2_Err_Fram_1.v				:= NOT( GVL.IIVD.S_TmOut_Kapi_Hatalari_1_0X230 OR GVL.IIVD.Z_Dr2_Err_Fram_1.RangeExcd OR GVL.IIVD.Z_Dr2_Err_Fram_1.e OR GVL.IIVD.Z_Dr2_Err_Fram_1.na) ;
GVL.IIVD.Z_Dr2_Err_Fram_1.x				:= 
(*SELECT 1 : Is data valid ?*)				SEL(GVL.IIVD.Z_Dr2_Err_Fram_1.v,
(*DEFAULT value assigment*)					0,
(*Transmission is VALID*)					Raw_Z_Dr2_Err_Fram_1);
{endregion}
{region " SIGNAL AREA : NAME->Z_Dr2_Err_Fram_2 LENGTH->8 STARTBIT :40"}
Raw_Z_Dr2_Err_Fram_2					:= _FB_CanRx_Message_230.X_Byte_5;
GVL.IIVD.Z_Dr2_Err_Fram_2.e				:= (Raw_Z_Dr2_Err_Fram_2 > 16#FD) AND (Raw_Z_Dr2_Err_Fram_2 < 16#FF);
GVL.IIVD.Z_Dr2_Err_Fram_2.na			:= (Raw_Z_Dr2_Err_Fram_2 = 16#FF);
GVL.IIVD.Z_Dr2_Err_Fram_2.RangeExcd		:= NOT ((Raw_Z_Dr2_Err_Fram_2 >= 0) AND (Raw_Z_Dr2_Err_Fram_2 <= 255));
GVL.IIVD.Z_Dr2_Err_Fram_2.v				:= NOT( GVL.IIVD.S_TmOut_Kapi_Hatalari_1_0X230 OR GVL.IIVD.Z_Dr2_Err_Fram_2.RangeExcd OR GVL.IIVD.Z_Dr2_Err_Fram_2.e OR GVL.IIVD.Z_Dr2_Err_Fram_2.na) ;
GVL.IIVD.Z_Dr2_Err_Fram_2.x				:= 
(*SELECT 1 : Is data valid ?*)				SEL(GVL.IIVD.Z_Dr2_Err_Fram_2.v,
(*DEFAULT value assigment*)					0,
(*Transmission is VALID*)					Raw_Z_Dr2_Err_Fram_2);
{endregion}
{region " SIGNAL AREA : NAME->Z_Dr2_Err_Fram_3 LENGTH->8 STARTBIT :48"}
Raw_Z_Dr2_Err_Fram_3					:= _FB_CanRx_Message_230.X_Byte_6;
GVL.IIVD.Z_Dr2_Err_Fram_3.e				:= (Raw_Z_Dr2_Err_Fram_3 > 16#FD) AND (Raw_Z_Dr2_Err_Fram_3 < 16#FF);
GVL.IIVD.Z_Dr2_Err_Fram_3.na			:= (Raw_Z_Dr2_Err_Fram_3 = 16#FF);
GVL.IIVD.Z_Dr2_Err_Fram_3.RangeExcd		:= NOT ((Raw_Z_Dr2_Err_Fram_3 >= 0) AND (Raw_Z_Dr2_Err_Fram_3 <= 255));
GVL.IIVD.Z_Dr2_Err_Fram_3.v				:= NOT( GVL.IIVD.S_TmOut_Kapi_Hatalari_1_0X230 OR GVL.IIVD.Z_Dr2_Err_Fram_3.RangeExcd OR GVL.IIVD.Z_Dr2_Err_Fram_3.e OR GVL.IIVD.Z_Dr2_Err_Fram_3.na) ;
GVL.IIVD.Z_Dr2_Err_Fram_3.x				:= 
(*SELECT 1 : Is data valid ?*)				SEL(GVL.IIVD.Z_Dr2_Err_Fram_3.v,
(*DEFAULT value assigment*)					0,
(*Transmission is VALID*)					Raw_Z_Dr2_Err_Fram_3);
{endregion}
{endregion}

{region " MESSAGE AREA :Kapi_Hatalari_2- ID:231"}

_FB_CanRx_Message_231 (		C_Enable	:= GVL.IIVD.S_CAN_Init,
     						Obj_CAN		:= ADR(GVL.IC.Obj_CAN0),
     						X_MsgID		:= 16#231,
     						Tm_MsgTmOut	:= TIME#2500MS,
     						S_Extended	:= 0,
     						S_ER_TmOut	=> GVL.IIVD.S_TmOut_Kapi_Hatalari_2_0X231);

{region " SIGNAL AREA : NAME->Z_Dr3_Err_Fram_1 LENGTH->8 STARTBIT :0"}
Raw_Z_Dr3_Err_Fram_1					:= _FB_CanRx_Message_231.X_Byte_0;
GVL.IIVD.Z_Dr3_Err_Fram_1.e				:= (Raw_Z_Dr3_Err_Fram_1 > 16#FD) AND (Raw_Z_Dr3_Err_Fram_1 < 16#FF);
GVL.IIVD.Z_Dr3_Err_Fram_1.na			:= (Raw_Z_Dr3_Err_Fram_1 = 16#FF);
GVL.IIVD.Z_Dr3_Err_Fram_1.RangeExcd		:= NOT ((Raw_Z_Dr3_Err_Fram_1 >= 0) AND (Raw_Z_Dr3_Err_Fram_1 <= 255));
GVL.IIVD.Z_Dr3_Err_Fram_1.v				:= NOT( GVL.IIVD.S_TmOut_Kapi_Hatalari_2_0X231 OR GVL.IIVD.Z_Dr3_Err_Fram_1.RangeExcd OR GVL.IIVD.Z_Dr3_Err_Fram_1.e OR GVL.IIVD.Z_Dr3_Err_Fram_1.na) ;
GVL.IIVD.Z_Dr3_Err_Fram_1.x				:= 
(*SELECT 1 : Is data valid ?*)				SEL(GVL.IIVD.Z_Dr3_Err_Fram_1.v,
(*DEFAULT value assigment*)					0,
(*Transmission is VALID*)					Raw_Z_Dr3_Err_Fram_1);
{endregion}
{region " SIGNAL AREA : NAME->Z_Dr3_Err_Fram_2 LENGTH->8 STARTBIT :8"}
Raw_Z_Dr3_Err_Fram_2					:= _FB_CanRx_Message_231.X_Byte_1;
GVL.IIVD.Z_Dr3_Err_Fram_2.e				:= (Raw_Z_Dr3_Err_Fram_2 > 16#FD) AND (Raw_Z_Dr3_Err_Fram_2 < 16#FF);
GVL.IIVD.Z_Dr3_Err_Fram_2.na			:= (Raw_Z_Dr3_Err_Fram_2 = 16#FF);
GVL.IIVD.Z_Dr3_Err_Fram_2.RangeExcd		:= NOT ((Raw_Z_Dr3_Err_Fram_2 >= 0) AND (Raw_Z_Dr3_Err_Fram_2 <= 255));
GVL.IIVD.Z_Dr3_Err_Fram_2.v				:= NOT( GVL.IIVD.S_TmOut_Kapi_Hatalari_2_0X231 OR GVL.IIVD.Z_Dr3_Err_Fram_2.RangeExcd OR GVL.IIVD.Z_Dr3_Err_Fram_2.e OR GVL.IIVD.Z_Dr3_Err_Fram_2.na) ;
GVL.IIVD.Z_Dr3_Err_Fram_2.x				:= 
(*SELECT 1 : Is data valid ?*)				SEL(GVL.IIVD.Z_Dr3_Err_Fram_2.v,
(*DEFAULT value assigment*)					0,
(*Transmission is VALID*)					Raw_Z_Dr3_Err_Fram_2);
{endregion}
{region " SIGNAL AREA : NAME->Z_Dr3_Err_Fram_3 LENGTH->8 STARTBIT :16"}
Raw_Z_Dr3_Err_Fram_3					:= _FB_CanRx_Message_231.X_Byte_2;
GVL.IIVD.Z_Dr3_Err_Fram_3.e				:= (Raw_Z_Dr3_Err_Fram_3 > 16#FD) AND (Raw_Z_Dr3_Err_Fram_3 < 16#FF);
GVL.IIVD.Z_Dr3_Err_Fram_3.na			:= (Raw_Z_Dr3_Err_Fram_3 = 16#FF);
GVL.IIVD.Z_Dr3_Err_Fram_3.RangeExcd		:= NOT ((Raw_Z_Dr3_Err_Fram_3 >= 0) AND (Raw_Z_Dr3_Err_Fram_3 <= 255));
GVL.IIVD.Z_Dr3_Err_Fram_3.v				:= NOT( GVL.IIVD.S_TmOut_Kapi_Hatalari_2_0X231 OR GVL.IIVD.Z_Dr3_Err_Fram_3.RangeExcd OR GVL.IIVD.Z_Dr3_Err_Fram_3.e OR GVL.IIVD.Z_Dr3_Err_Fram_3.na) ;
GVL.IIVD.Z_Dr3_Err_Fram_3.x				:= 
(*SELECT 1 : Is data valid ?*)				SEL(GVL.IIVD.Z_Dr3_Err_Fram_3.v,
(*DEFAULT value assigment*)					0,
(*Transmission is VALID*)					Raw_Z_Dr3_Err_Fram_3);
{endregion}
{region " SIGNAL AREA : NAME->Z_Dr4_Err_Fram_1 LENGTH->8 STARTBIT :32"}
Raw_Z_Dr4_Err_Fram_1					:= _FB_CanRx_Message_231.X_Byte_4;
GVL.IIVD.Z_Dr4_Err_Fram_1.e				:= (Raw_Z_Dr4_Err_Fram_1 > 16#FD) AND (Raw_Z_Dr4_Err_Fram_1 < 16#FF);
GVL.IIVD.Z_Dr4_Err_Fram_1.na			:= (Raw_Z_Dr4_Err_Fram_1 = 16#FF);
GVL.IIVD.Z_Dr4_Err_Fram_1.RangeExcd		:= NOT ((Raw_Z_Dr4_Err_Fram_1 >= 0) AND (Raw_Z_Dr4_Err_Fram_1 <= 255));
GVL.IIVD.Z_Dr4_Err_Fram_1.v				:= NOT( GVL.IIVD.S_TmOut_Kapi_Hatalari_2_0X231 OR GVL.IIVD.Z_Dr4_Err_Fram_1.RangeExcd OR GVL.IIVD.Z_Dr4_Err_Fram_1.e OR GVL.IIVD.Z_Dr4_Err_Fram_1.na) ;
GVL.IIVD.Z_Dr4_Err_Fram_1.x				:= 
(*SELECT 1 : Is data valid ?*)				SEL(GVL.IIVD.Z_Dr4_Err_Fram_1.v,
(*DEFAULT value assigment*)					0,
(*Transmission is VALID*)					Raw_Z_Dr4_Err_Fram_1);
{endregion}
{region " SIGNAL AREA : NAME->Z_Dr4_Err_Fram_2 LENGTH->8 STARTBIT :40"}
Raw_Z_Dr4_Err_Fram_2					:= _FB_CanRx_Message_231.X_Byte_5;
GVL.IIVD.Z_Dr4_Err_Fram_2.e				:= (Raw_Z_Dr4_Err_Fram_2 > 16#FD) AND (Raw_Z_Dr4_Err_Fram_2 < 16#FF);
GVL.IIVD.Z_Dr4_Err_Fram_2.na			:= (Raw_Z_Dr4_Err_Fram_2 = 16#FF);
GVL.IIVD.Z_Dr4_Err_Fram_2.RangeExcd		:= NOT ((Raw_Z_Dr4_Err_Fram_2 >= 0) AND (Raw_Z_Dr4_Err_Fram_2 <= 255));
GVL.IIVD.Z_Dr4_Err_Fram_2.v				:= NOT( GVL.IIVD.S_TmOut_Kapi_Hatalari_2_0X231 OR GVL.IIVD.Z_Dr4_Err_Fram_2.RangeExcd OR GVL.IIVD.Z_Dr4_Err_Fram_2.e OR GVL.IIVD.Z_Dr4_Err_Fram_2.na) ;
GVL.IIVD.Z_Dr4_Err_Fram_2.x				:= 
(*SELECT 1 : Is data valid ?*)				SEL(GVL.IIVD.Z_Dr4_Err_Fram_2.v,
(*DEFAULT value assigment*)					0,
(*Transmission is VALID*)					Raw_Z_Dr4_Err_Fram_2);
{endregion}
{region " SIGNAL AREA : NAME->Z_Dr4_Err_Fram_3 LENGTH->8 STARTBIT :48"}
Raw_Z_Dr4_Err_Fram_3					:= _FB_CanRx_Message_231.X_Byte_6;
GVL.IIVD.Z_Dr4_Err_Fram_3.e				:= (Raw_Z_Dr4_Err_Fram_3 > 16#FD) AND (Raw_Z_Dr4_Err_Fram_3 < 16#FF);
GVL.IIVD.Z_Dr4_Err_Fram_3.na			:= (Raw_Z_Dr4_Err_Fram_3 = 16#FF);
GVL.IIVD.Z_Dr4_Err_Fram_3.RangeExcd		:= NOT ((Raw_Z_Dr4_Err_Fram_3 >= 0) AND (Raw_Z_Dr4_Err_Fram_3 <= 255));
GVL.IIVD.Z_Dr4_Err_Fram_3.v				:= NOT( GVL.IIVD.S_TmOut_Kapi_Hatalari_2_0X231 OR GVL.IIVD.Z_Dr4_Err_Fram_3.RangeExcd OR GVL.IIVD.Z_Dr4_Err_Fram_3.e OR GVL.IIVD.Z_Dr4_Err_Fram_3.na) ;
GVL.IIVD.Z_Dr4_Err_Fram_3.x				:= 
(*SELECT 1 : Is data valid ?*)				SEL(GVL.IIVD.Z_Dr4_Err_Fram_3.v,
(*DEFAULT value assigment*)					0,
(*Transmission is VALID*)					Raw_Z_Dr4_Err_Fram_3);
{endregion}
{endregion}

{region " MESSAGE AREA :Kapi_Hatalari_3- ID:232"}

_FB_CanRx_Message_232 (		C_Enable	:= GVL.IIVD.S_CAN_Init,
     						Obj_CAN		:= ADR(GVL.IC.Obj_CAN0),
     						X_MsgID		:= 16#232,
     						Tm_MsgTmOut	:= TIME#2500MS,
     						S_Extended	:= 0,
     						S_ER_TmOut	=> GVL.IIVD.S_TmOut_Kapi_Hatalari_3_0X232);

{region " SIGNAL AREA : NAME->Z_Dr5_Err_Fram_1 LENGTH->8 STARTBIT :0"}
Raw_Z_Dr5_Err_Fram_1					:= _FB_CanRx_Message_232.X_Byte_0;
GVL.IIVD.Z_Dr5_Err_Fram_1.e				:= (Raw_Z_Dr5_Err_Fram_1 > 16#FD) AND (Raw_Z_Dr5_Err_Fram_1 < 16#FF);
GVL.IIVD.Z_Dr5_Err_Fram_1.na			:= (Raw_Z_Dr5_Err_Fram_1 = 16#FF);
GVL.IIVD.Z_Dr5_Err_Fram_1.RangeExcd		:= NOT ((Raw_Z_Dr5_Err_Fram_1 >= 0) AND (Raw_Z_Dr5_Err_Fram_1 <= 255));
GVL.IIVD.Z_Dr5_Err_Fram_1.v				:= NOT( GVL.IIVD.S_TmOut_Kapi_Hatalari_3_0X232 OR GVL.IIVD.Z_Dr5_Err_Fram_1.RangeExcd OR GVL.IIVD.Z_Dr5_Err_Fram_1.e OR GVL.IIVD.Z_Dr5_Err_Fram_1.na) ;
GVL.IIVD.Z_Dr5_Err_Fram_1.x				:= 
(*SELECT 1 : Is data valid ?*)				SEL(GVL.IIVD.Z_Dr5_Err_Fram_1.v,
(*DEFAULT value assigment*)					0,
(*Transmission is VALID*)					Raw_Z_Dr5_Err_Fram_1);
{endregion}
{region " SIGNAL AREA : NAME->Z_Dr5_Err_Fram_2 LENGTH->8 STARTBIT :8"}
Raw_Z_Dr5_Err_Fram_2					:= _FB_CanRx_Message_232.X_Byte_1;
GVL.IIVD.Z_Dr5_Err_Fram_2.e				:= (Raw_Z_Dr5_Err_Fram_2 > 16#FD) AND (Raw_Z_Dr5_Err_Fram_2 < 16#FF);
GVL.IIVD.Z_Dr5_Err_Fram_2.na			:= (Raw_Z_Dr5_Err_Fram_2 = 16#FF);
GVL.IIVD.Z_Dr5_Err_Fram_2.RangeExcd		:= NOT ((Raw_Z_Dr5_Err_Fram_2 >= 0) AND (Raw_Z_Dr5_Err_Fram_2 <= 255));
GVL.IIVD.Z_Dr5_Err_Fram_2.v				:= NOT( GVL.IIVD.S_TmOut_Kapi_Hatalari_3_0X232 OR GVL.IIVD.Z_Dr5_Err_Fram_2.RangeExcd OR GVL.IIVD.Z_Dr5_Err_Fram_2.e OR GVL.IIVD.Z_Dr5_Err_Fram_2.na) ;
GVL.IIVD.Z_Dr5_Err_Fram_2.x				:= 
(*SELECT 1 : Is data valid ?*)				SEL(GVL.IIVD.Z_Dr5_Err_Fram_2.v,
(*DEFAULT value assigment*)					0,
(*Transmission is VALID*)					Raw_Z_Dr5_Err_Fram_2);
{endregion}
{region " SIGNAL AREA : NAME->Z_Dr5_Err_Fram_3 LENGTH->8 STARTBIT :16"}
Raw_Z_Dr5_Err_Fram_3					:= _FB_CanRx_Message_232.X_Byte_2;
GVL.IIVD.Z_Dr5_Err_Fram_3.e				:= (Raw_Z_Dr5_Err_Fram_3 > 16#FD) AND (Raw_Z_Dr5_Err_Fram_3 < 16#FF);
GVL.IIVD.Z_Dr5_Err_Fram_3.na			:= (Raw_Z_Dr5_Err_Fram_3 = 16#FF);
GVL.IIVD.Z_Dr5_Err_Fram_3.RangeExcd		:= NOT ((Raw_Z_Dr5_Err_Fram_3 >= 0) AND (Raw_Z_Dr5_Err_Fram_3 <= 255));
GVL.IIVD.Z_Dr5_Err_Fram_3.v				:= NOT( GVL.IIVD.S_TmOut_Kapi_Hatalari_3_0X232 OR GVL.IIVD.Z_Dr5_Err_Fram_3.RangeExcd OR GVL.IIVD.Z_Dr5_Err_Fram_3.e OR GVL.IIVD.Z_Dr5_Err_Fram_3.na) ;
GVL.IIVD.Z_Dr5_Err_Fram_3.x				:= 
(*SELECT 1 : Is data valid ?*)				SEL(GVL.IIVD.Z_Dr5_Err_Fram_3.v,
(*DEFAULT value assigment*)					0,
(*Transmission is VALID*)					Raw_Z_Dr5_Err_Fram_3);
{endregion}
{region " SIGNAL AREA : NAME->Z_Dr6_Err_Fram_1 LENGTH->8 STARTBIT :32"}
Raw_Z_Dr6_Err_Fram_1					:= _FB_CanRx_Message_232.X_Byte_4;
GVL.IIVD.Z_Dr6_Err_Fram_1.e				:= (Raw_Z_Dr6_Err_Fram_1 > 16#FD) AND (Raw_Z_Dr6_Err_Fram_1 < 16#FF);
GVL.IIVD.Z_Dr6_Err_Fram_1.na			:= (Raw_Z_Dr6_Err_Fram_1 = 16#FF);
GVL.IIVD.Z_Dr6_Err_Fram_1.RangeExcd		:= NOT ((Raw_Z_Dr6_Err_Fram_1 >= 0) AND (Raw_Z_Dr6_Err_Fram_1 <= 255));
GVL.IIVD.Z_Dr6_Err_Fram_1.v				:= NOT( GVL.IIVD.S_TmOut_Kapi_Hatalari_3_0X232 OR GVL.IIVD.Z_Dr6_Err_Fram_1.RangeExcd OR GVL.IIVD.Z_Dr6_Err_Fram_1.e OR GVL.IIVD.Z_Dr6_Err_Fram_1.na) ;
GVL.IIVD.Z_Dr6_Err_Fram_1.x				:= 
(*SELECT 1 : Is data valid ?*)				SEL(GVL.IIVD.Z_Dr6_Err_Fram_1.v,
(*DEFAULT value assigment*)					0,
(*Transmission is VALID*)					Raw_Z_Dr6_Err_Fram_1);
{endregion}
{region " SIGNAL AREA : NAME->Z_Dr6_Err_Fram_2 LENGTH->8 STARTBIT :40"}
Raw_Z_Dr6_Err_Fram_2					:= _FB_CanRx_Message_232.X_Byte_5;
GVL.IIVD.Z_Dr6_Err_Fram_2.e				:= (Raw_Z_Dr6_Err_Fram_2 > 16#FD) AND (Raw_Z_Dr6_Err_Fram_2 < 16#FF);
GVL.IIVD.Z_Dr6_Err_Fram_2.na			:= (Raw_Z_Dr6_Err_Fram_2 = 16#FF);
GVL.IIVD.Z_Dr6_Err_Fram_2.RangeExcd		:= NOT ((Raw_Z_Dr6_Err_Fram_2 >= 0) AND (Raw_Z_Dr6_Err_Fram_2 <= 255));
GVL.IIVD.Z_Dr6_Err_Fram_2.v				:= NOT( GVL.IIVD.S_TmOut_Kapi_Hatalari_3_0X232 OR GVL.IIVD.Z_Dr6_Err_Fram_2.RangeExcd OR GVL.IIVD.Z_Dr6_Err_Fram_2.e OR GVL.IIVD.Z_Dr6_Err_Fram_2.na) ;
GVL.IIVD.Z_Dr6_Err_Fram_2.x				:= 
(*SELECT 1 : Is data valid ?*)				SEL(GVL.IIVD.Z_Dr6_Err_Fram_2.v,
(*DEFAULT value assigment*)					0,
(*Transmission is VALID*)					Raw_Z_Dr6_Err_Fram_2);
{endregion}
{region " SIGNAL AREA : NAME->Z_Dr6_Err_Fram_3 LENGTH->8 STARTBIT :48"}
Raw_Z_Dr6_Err_Fram_3					:= _FB_CanRx_Message_232.X_Byte_6;
GVL.IIVD.Z_Dr6_Err_Fram_3.e				:= (Raw_Z_Dr6_Err_Fram_3 > 16#FD) AND (Raw_Z_Dr6_Err_Fram_3 < 16#FF);
GVL.IIVD.Z_Dr6_Err_Fram_3.na			:= (Raw_Z_Dr6_Err_Fram_3 = 16#FF);
GVL.IIVD.Z_Dr6_Err_Fram_3.RangeExcd		:= NOT ((Raw_Z_Dr6_Err_Fram_3 >= 0) AND (Raw_Z_Dr6_Err_Fram_3 <= 255));
GVL.IIVD.Z_Dr6_Err_Fram_3.v				:= NOT( GVL.IIVD.S_TmOut_Kapi_Hatalari_3_0X232 OR GVL.IIVD.Z_Dr6_Err_Fram_3.RangeExcd OR GVL.IIVD.Z_Dr6_Err_Fram_3.e OR GVL.IIVD.Z_Dr6_Err_Fram_3.na) ;
GVL.IIVD.Z_Dr6_Err_Fram_3.x				:= 
(*SELECT 1 : Is data valid ?*)				SEL(GVL.IIVD.Z_Dr6_Err_Fram_3.v,
(*DEFAULT value assigment*)					0,
(*Transmission is VALID*)					Raw_Z_Dr6_Err_Fram_3);
{endregion}
{endregion}

{region " MESSAGE AREA :Kapi_Hatalari_4- ID:233"}

_FB_CanRx_Message_233 (		C_Enable	:= GVL.IIVD.S_CAN_Init,
     						Obj_CAN		:= ADR(GVL.IC.Obj_CAN0),
     						X_MsgID		:= 16#233,
     						Tm_MsgTmOut	:= TIME#2500MS,
     						S_Extended	:= 0,
     						S_ER_TmOut	=> GVL.IIVD.S_TmOut_Kapi_Hatalari_4_0X233);

{region " SIGNAL AREA : NAME->Z_Dr7_Err_Fram_1 LENGTH->8 STARTBIT :0"}
Raw_Z_Dr7_Err_Fram_1					:= _FB_CanRx_Message_233.X_Byte_0;
GVL.IIVD.Z_Dr7_Err_Fram_1.e				:= (Raw_Z_Dr7_Err_Fram_1 > 16#FD) AND (Raw_Z_Dr7_Err_Fram_1 < 16#FF);
GVL.IIVD.Z_Dr7_Err_Fram_1.na			:= (Raw_Z_Dr7_Err_Fram_1 = 16#FF);
GVL.IIVD.Z_Dr7_Err_Fram_1.RangeExcd		:= NOT ((Raw_Z_Dr7_Err_Fram_1 >= 0) AND (Raw_Z_Dr7_Err_Fram_1 <= 255));
GVL.IIVD.Z_Dr7_Err_Fram_1.v				:= NOT( GVL.IIVD.S_TmOut_Kapi_Hatalari_4_0X233 OR GVL.IIVD.Z_Dr7_Err_Fram_1.RangeExcd OR GVL.IIVD.Z_Dr7_Err_Fram_1.e OR GVL.IIVD.Z_Dr7_Err_Fram_1.na) ;
GVL.IIVD.Z_Dr7_Err_Fram_1.x				:= 
(*SELECT 1 : Is data valid ?*)				SEL(GVL.IIVD.Z_Dr7_Err_Fram_1.v,
(*DEFAULT value assigment*)					0,
(*Transmission is VALID*)					Raw_Z_Dr7_Err_Fram_1);
{endregion}
{region " SIGNAL AREA : NAME->Z_Dr7_Err_Fram_2 LENGTH->8 STARTBIT :8"}
Raw_Z_Dr7_Err_Fram_2					:= _FB_CanRx_Message_233.X_Byte_1;
GVL.IIVD.Z_Dr7_Err_Fram_2.e				:= (Raw_Z_Dr7_Err_Fram_2 > 16#FD) AND (Raw_Z_Dr7_Err_Fram_2 < 16#FF);
GVL.IIVD.Z_Dr7_Err_Fram_2.na			:= (Raw_Z_Dr7_Err_Fram_2 = 16#FF);
GVL.IIVD.Z_Dr7_Err_Fram_2.RangeExcd		:= NOT ((Raw_Z_Dr7_Err_Fram_2 >= 0) AND (Raw_Z_Dr7_Err_Fram_2 <= 255));
GVL.IIVD.Z_Dr7_Err_Fram_2.v				:= NOT( GVL.IIVD.S_TmOut_Kapi_Hatalari_4_0X233 OR GVL.IIVD.Z_Dr7_Err_Fram_2.RangeExcd OR GVL.IIVD.Z_Dr7_Err_Fram_2.e OR GVL.IIVD.Z_Dr7_Err_Fram_2.na) ;
GVL.IIVD.Z_Dr7_Err_Fram_2.x				:= 
(*SELECT 1 : Is data valid ?*)				SEL(GVL.IIVD.Z_Dr7_Err_Fram_2.v,
(*DEFAULT value assigment*)					0,
(*Transmission is VALID*)					Raw_Z_Dr7_Err_Fram_2);
{endregion}
{region " SIGNAL AREA : NAME->Z_Dr7_Err_Fram_3 LENGTH->8 STARTBIT :16"}
Raw_Z_Dr7_Err_Fram_3					:= _FB_CanRx_Message_233.X_Byte_2;
GVL.IIVD.Z_Dr7_Err_Fram_3.e				:= (Raw_Z_Dr7_Err_Fram_3 > 16#FD) AND (Raw_Z_Dr7_Err_Fram_3 < 16#FF);
GVL.IIVD.Z_Dr7_Err_Fram_3.na			:= (Raw_Z_Dr7_Err_Fram_3 = 16#FF);
GVL.IIVD.Z_Dr7_Err_Fram_3.RangeExcd		:= NOT ((Raw_Z_Dr7_Err_Fram_3 >= 0) AND (Raw_Z_Dr7_Err_Fram_3 <= 255));
GVL.IIVD.Z_Dr7_Err_Fram_3.v				:= NOT( GVL.IIVD.S_TmOut_Kapi_Hatalari_4_0X233 OR GVL.IIVD.Z_Dr7_Err_Fram_3.RangeExcd OR GVL.IIVD.Z_Dr7_Err_Fram_3.e OR GVL.IIVD.Z_Dr7_Err_Fram_3.na) ;
GVL.IIVD.Z_Dr7_Err_Fram_3.x				:= 
(*SELECT 1 : Is data valid ?*)				SEL(GVL.IIVD.Z_Dr7_Err_Fram_3.v,
(*DEFAULT value assigment*)					0,
(*Transmission is VALID*)					Raw_Z_Dr7_Err_Fram_3);
{endregion}
{region " SIGNAL AREA : NAME->Z_Dr8_Err_Fram_1 LENGTH->8 STARTBIT :32"}
Raw_Z_Dr8_Err_Fram_1					:= _FB_CanRx_Message_233.X_Byte_4;
GVL.IIVD.Z_Dr8_Err_Fram_1.e				:= (Raw_Z_Dr8_Err_Fram_1 > 16#FD) AND (Raw_Z_Dr8_Err_Fram_1 < 16#FF);
GVL.IIVD.Z_Dr8_Err_Fram_1.na			:= (Raw_Z_Dr8_Err_Fram_1 = 16#FF);
GVL.IIVD.Z_Dr8_Err_Fram_1.RangeExcd		:= NOT ((Raw_Z_Dr8_Err_Fram_1 >= 0) AND (Raw_Z_Dr8_Err_Fram_1 <= 255));
GVL.IIVD.Z_Dr8_Err_Fram_1.v				:= NOT( GVL.IIVD.S_TmOut_Kapi_Hatalari_4_0X233 OR GVL.IIVD.Z_Dr8_Err_Fram_1.RangeExcd OR GVL.IIVD.Z_Dr8_Err_Fram_1.e OR GVL.IIVD.Z_Dr8_Err_Fram_1.na) ;
GVL.IIVD.Z_Dr8_Err_Fram_1.x				:= 
(*SELECT 1 : Is data valid ?*)				SEL(GVL.IIVD.Z_Dr8_Err_Fram_1.v,
(*DEFAULT value assigment*)					0,
(*Transmission is VALID*)					Raw_Z_Dr8_Err_Fram_1);
{endregion}
{region " SIGNAL AREA : NAME->Z_Dr8_Err_Fram_2 LENGTH->8 STARTBIT :40"}
Raw_Z_Dr8_Err_Fram_2					:= _FB_CanRx_Message_233.X_Byte_5;
GVL.IIVD.Z_Dr8_Err_Fram_2.e				:= (Raw_Z_Dr8_Err_Fram_2 > 16#FD) AND (Raw_Z_Dr8_Err_Fram_2 < 16#FF);
GVL.IIVD.Z_Dr8_Err_Fram_2.na			:= (Raw_Z_Dr8_Err_Fram_2 = 16#FF);
GVL.IIVD.Z_Dr8_Err_Fram_2.RangeExcd		:= NOT ((Raw_Z_Dr8_Err_Fram_2 >= 0) AND (Raw_Z_Dr8_Err_Fram_2 <= 255));
GVL.IIVD.Z_Dr8_Err_Fram_2.v				:= NOT( GVL.IIVD.S_TmOut_Kapi_Hatalari_4_0X233 OR GVL.IIVD.Z_Dr8_Err_Fram_2.RangeExcd OR GVL.IIVD.Z_Dr8_Err_Fram_2.e OR GVL.IIVD.Z_Dr8_Err_Fram_2.na) ;
GVL.IIVD.Z_Dr8_Err_Fram_2.x				:= 
(*SELECT 1 : Is data valid ?*)				SEL(GVL.IIVD.Z_Dr8_Err_Fram_2.v,
(*DEFAULT value assigment*)					0,
(*Transmission is VALID*)					Raw_Z_Dr8_Err_Fram_2);
{endregion}
{region " SIGNAL AREA : NAME->Z_Dr8_Err_Fram_3 LENGTH->8 STARTBIT :48"}
Raw_Z_Dr8_Err_Fram_3					:= _FB_CanRx_Message_233.X_Byte_6;
GVL.IIVD.Z_Dr8_Err_Fram_3.e				:= (Raw_Z_Dr8_Err_Fram_3 > 16#FD) AND (Raw_Z_Dr8_Err_Fram_3 < 16#FF);
GVL.IIVD.Z_Dr8_Err_Fram_3.na			:= (Raw_Z_Dr8_Err_Fram_3 = 16#FF);
GVL.IIVD.Z_Dr8_Err_Fram_3.RangeExcd		:= NOT ((Raw_Z_Dr8_Err_Fram_3 >= 0) AND (Raw_Z_Dr8_Err_Fram_3 <= 255));
GVL.IIVD.Z_Dr8_Err_Fram_3.v				:= NOT( GVL.IIVD.S_TmOut_Kapi_Hatalari_4_0X233 OR GVL.IIVD.Z_Dr8_Err_Fram_3.RangeExcd OR GVL.IIVD.Z_Dr8_Err_Fram_3.e OR GVL.IIVD.Z_Dr8_Err_Fram_3.na) ;
GVL.IIVD.Z_Dr8_Err_Fram_3.x				:= 
(*SELECT 1 : Is data valid ?*)				SEL(GVL.IIVD.Z_Dr8_Err_Fram_3.v,
(*DEFAULT value assigment*)					0,
(*Transmission is VALID*)					Raw_Z_Dr8_Err_Fram_3);
{endregion}
{endregion}

{region " MESSAGE AREA :Kapi_Hatalari_5- ID:234"}

_FB_CanRx_Message_234 (		C_Enable	:= GVL.IIVD.S_CAN_Init,
     						Obj_CAN		:= ADR(GVL.IC.Obj_CAN0),
     						X_MsgID		:= 16#234,
     						Tm_MsgTmOut	:= TIME#2500MS,
     						S_Extended	:= 0,
     						S_ER_TmOut	=> GVL.IIVD.S_TmOut_Kapi_Hatalari_5_0X234);

{region " SIGNAL AREA : NAME->Z_Dr9_Err_Fram_1 LENGTH->8 STARTBIT :0"}
Raw_Z_Dr9_Err_Fram_1					:= _FB_CanRx_Message_234.X_Byte_0;
GVL.IIVD.Z_Dr9_Err_Fram_1.e				:= (Raw_Z_Dr9_Err_Fram_1 > 16#FD) AND (Raw_Z_Dr9_Err_Fram_1 < 16#FF);
GVL.IIVD.Z_Dr9_Err_Fram_1.na			:= (Raw_Z_Dr9_Err_Fram_1 = 16#FF);
GVL.IIVD.Z_Dr9_Err_Fram_1.RangeExcd		:= NOT ((Raw_Z_Dr9_Err_Fram_1 >= 0) AND (Raw_Z_Dr9_Err_Fram_1 <= 255));
GVL.IIVD.Z_Dr9_Err_Fram_1.v				:= NOT( GVL.IIVD.S_TmOut_Kapi_Hatalari_5_0X234 OR GVL.IIVD.Z_Dr9_Err_Fram_1.RangeExcd OR GVL.IIVD.Z_Dr9_Err_Fram_1.e OR GVL.IIVD.Z_Dr9_Err_Fram_1.na) ;
GVL.IIVD.Z_Dr9_Err_Fram_1.x				:= 
(*SELECT 1 : Is data valid ?*)				SEL(GVL.IIVD.Z_Dr9_Err_Fram_1.v,
(*DEFAULT value assigment*)					0,
(*Transmission is VALID*)					Raw_Z_Dr9_Err_Fram_1);
{endregion}
{region " SIGNAL AREA : NAME->Z_Dr9_Err_Fram_2 LENGTH->8 STARTBIT :8"}
Raw_Z_Dr9_Err_Fram_2					:= _FB_CanRx_Message_234.X_Byte_1;
GVL.IIVD.Z_Dr9_Err_Fram_2.e				:= (Raw_Z_Dr9_Err_Fram_2 > 16#FD) AND (Raw_Z_Dr9_Err_Fram_2 < 16#FF);
GVL.IIVD.Z_Dr9_Err_Fram_2.na			:= (Raw_Z_Dr9_Err_Fram_2 = 16#FF);
GVL.IIVD.Z_Dr9_Err_Fram_2.RangeExcd		:= NOT ((Raw_Z_Dr9_Err_Fram_2 >= 0) AND (Raw_Z_Dr9_Err_Fram_2 <= 255));
GVL.IIVD.Z_Dr9_Err_Fram_2.v				:= NOT( GVL.IIVD.S_TmOut_Kapi_Hatalari_5_0X234 OR GVL.IIVD.Z_Dr9_Err_Fram_2.RangeExcd OR GVL.IIVD.Z_Dr9_Err_Fram_2.e OR GVL.IIVD.Z_Dr9_Err_Fram_2.na) ;
GVL.IIVD.Z_Dr9_Err_Fram_2.x				:= 
(*SELECT 1 : Is data valid ?*)				SEL(GVL.IIVD.Z_Dr9_Err_Fram_2.v,
(*DEFAULT value assigment*)					0,
(*Transmission is VALID*)					Raw_Z_Dr9_Err_Fram_2);
{endregion}
{region " SIGNAL AREA : NAME->Z_Dr9_Err_Fram_3 LENGTH->8 STARTBIT :16"}
Raw_Z_Dr9_Err_Fram_3					:= _FB_CanRx_Message_234.X_Byte_2;
GVL.IIVD.Z_Dr9_Err_Fram_3.e				:= (Raw_Z_Dr9_Err_Fram_3 > 16#FD) AND (Raw_Z_Dr9_Err_Fram_3 < 16#FF);
GVL.IIVD.Z_Dr9_Err_Fram_3.na			:= (Raw_Z_Dr9_Err_Fram_3 = 16#FF);
GVL.IIVD.Z_Dr9_Err_Fram_3.RangeExcd		:= NOT ((Raw_Z_Dr9_Err_Fram_3 >= 0) AND (Raw_Z_Dr9_Err_Fram_3 <= 255));
GVL.IIVD.Z_Dr9_Err_Fram_3.v				:= NOT( GVL.IIVD.S_TmOut_Kapi_Hatalari_5_0X234 OR GVL.IIVD.Z_Dr9_Err_Fram_3.RangeExcd OR GVL.IIVD.Z_Dr9_Err_Fram_3.e OR GVL.IIVD.Z_Dr9_Err_Fram_3.na) ;
GVL.IIVD.Z_Dr9_Err_Fram_3.x				:= 
(*SELECT 1 : Is data valid ?*)				SEL(GVL.IIVD.Z_Dr9_Err_Fram_3.v,
(*DEFAULT value assigment*)					0,
(*Transmission is VALID*)					Raw_Z_Dr9_Err_Fram_3);
{endregion}
{endregion}

{region " MESSAGE AREA :Kapi_Durum_1- ID:235"}

_FB_CanRx_Message_Unpack_235 (		C_Enable	:= GVL.IIVD.S_CAN_Init,
     								Obj_CAN		:= ADR(GVL.IC.Obj_CAN0),
     								X_MsgID		:= 16#235,
     								Tm_MsgTmOut	:= TIME#2500MS,
     								S_Extended	:= 0,
     								S_ER_TmOut	=> GVL.IIVD.S_TmOut_Kapi_Durum_1_0X235);

{region " SIGNAL AREA : NAME->S_Dr1_Rhs_Leaf_Opng LENGTH->2 STARTBIT :0"}
GVL.IIVD.S_Dr1_Rhs_Leaf_Opng.v			:= NOT GVL.IIVD.S_TmOut_Kapi_Durum_1_0X235 AND NOT _FB_CanRx_Message_Unpack_235.S_Bit_1;
GVL.IIVD.S_Dr1_Rhs_Leaf_Opng.x			:= GVL.IIVD.S_Dr1_Rhs_Leaf_Opng.v AND _FB_CanRx_Message_Unpack_235.S_Bit_0;
GVL.IIVD.S_Dr1_Rhs_Leaf_Opng.e			:= _FB_CanRx_Message_Unpack_235.S_Bit_1 AND NOT _FB_CanRx_Message_Unpack_235.S_Bit_0 ;
GVL.IIVD.S_Dr1_Rhs_Leaf_Opng.na			:= _FB_CanRx_Message_Unpack_235.S_Bit_1 AND _FB_CanRx_Message_Unpack_235.S_Bit_0 ;
{endregion}
{region " SIGNAL AREA : NAME->S_Dr1_Rhs_Leaf_Clng LENGTH->2 STARTBIT :2"}
GVL.IIVD.S_Dr1_Rhs_Leaf_Clng.v			:= NOT GVL.IIVD.S_TmOut_Kapi_Durum_1_0X235 AND NOT _FB_CanRx_Message_Unpack_235.S_Bit_3;
GVL.IIVD.S_Dr1_Rhs_Leaf_Clng.x			:= GVL.IIVD.S_Dr1_Rhs_Leaf_Clng.v AND _FB_CanRx_Message_Unpack_235.S_Bit_2;
GVL.IIVD.S_Dr1_Rhs_Leaf_Clng.e			:= _FB_CanRx_Message_Unpack_235.S_Bit_3 AND NOT _FB_CanRx_Message_Unpack_235.S_Bit_2 ;
GVL.IIVD.S_Dr1_Rhs_Leaf_Clng.na			:= _FB_CanRx_Message_Unpack_235.S_Bit_3 AND _FB_CanRx_Message_Unpack_235.S_Bit_2 ;
{endregion}
{region " SIGNAL AREA : NAME->S_Dr1_Rhs_Leaf_Op LENGTH->2 STARTBIT :4"}
GVL.IIVD.S_Dr1_Rhs_Leaf_Op.v			:= NOT GVL.IIVD.S_TmOut_Kapi_Durum_1_0X235 AND NOT _FB_CanRx_Message_Unpack_235.S_Bit_5;
GVL.IIVD.S_Dr1_Rhs_Leaf_Op.x			:= GVL.IIVD.S_Dr1_Rhs_Leaf_Op.v AND _FB_CanRx_Message_Unpack_235.S_Bit_4;
GVL.IIVD.S_Dr1_Rhs_Leaf_Op.e			:= _FB_CanRx_Message_Unpack_235.S_Bit_5 AND NOT _FB_CanRx_Message_Unpack_235.S_Bit_4 ;
GVL.IIVD.S_Dr1_Rhs_Leaf_Op.na			:= _FB_CanRx_Message_Unpack_235.S_Bit_5 AND _FB_CanRx_Message_Unpack_235.S_Bit_4 ;
{endregion}
{region " SIGNAL AREA : NAME->S_Dr1_Rhs_Leaf_Cl LENGTH->2 STARTBIT :6"}
GVL.IIVD.S_Dr1_Rhs_Leaf_Cl.v			:= NOT GVL.IIVD.S_TmOut_Kapi_Durum_1_0X235 AND NOT _FB_CanRx_Message_Unpack_235.S_Bit_7;
GVL.IIVD.S_Dr1_Rhs_Leaf_Cl.x			:= GVL.IIVD.S_Dr1_Rhs_Leaf_Cl.v AND _FB_CanRx_Message_Unpack_235.S_Bit_6;
GVL.IIVD.S_Dr1_Rhs_Leaf_Cl.e			:= _FB_CanRx_Message_Unpack_235.S_Bit_7 AND NOT _FB_CanRx_Message_Unpack_235.S_Bit_6 ;
GVL.IIVD.S_Dr1_Rhs_Leaf_Cl.na			:= _FB_CanRx_Message_Unpack_235.S_Bit_7 AND _FB_CanRx_Message_Unpack_235.S_Bit_6 ;
{endregion}
{region " SIGNAL AREA : NAME->S_Dr1_Rhs_Leaf_Obs LENGTH->2 STARTBIT :8"}
GVL.IIVD.S_Dr1_Rhs_Leaf_Obs.v			:= NOT GVL.IIVD.S_TmOut_Kapi_Durum_1_0X235 AND NOT _FB_CanRx_Message_Unpack_235.S_Bit_9;
GVL.IIVD.S_Dr1_Rhs_Leaf_Obs.x			:= GVL.IIVD.S_Dr1_Rhs_Leaf_Obs.v AND _FB_CanRx_Message_Unpack_235.S_Bit_8;
GVL.IIVD.S_Dr1_Rhs_Leaf_Obs.e			:= _FB_CanRx_Message_Unpack_235.S_Bit_9 AND NOT _FB_CanRx_Message_Unpack_235.S_Bit_8 ;
GVL.IIVD.S_Dr1_Rhs_Leaf_Obs.na			:= _FB_CanRx_Message_Unpack_235.S_Bit_9 AND _FB_CanRx_Message_Unpack_235.S_Bit_8 ;
{endregion}
{region " SIGNAL AREA : NAME->S_Dr1_Lft_Leaf_Opng LENGTH->2 STARTBIT :10"}
GVL.IIVD.S_Dr1_Lft_Leaf_Opng.v			:= NOT GVL.IIVD.S_TmOut_Kapi_Durum_1_0X235 AND NOT _FB_CanRx_Message_Unpack_235.S_Bit_11;
GVL.IIVD.S_Dr1_Lft_Leaf_Opng.x			:= GVL.IIVD.S_Dr1_Lft_Leaf_Opng.v AND _FB_CanRx_Message_Unpack_235.S_Bit_10;
GVL.IIVD.S_Dr1_Lft_Leaf_Opng.e			:= _FB_CanRx_Message_Unpack_235.S_Bit_11 AND NOT _FB_CanRx_Message_Unpack_235.S_Bit_10 ;
GVL.IIVD.S_Dr1_Lft_Leaf_Opng.na			:= _FB_CanRx_Message_Unpack_235.S_Bit_11 AND _FB_CanRx_Message_Unpack_235.S_Bit_10 ;
{endregion}
{region " SIGNAL AREA : NAME->S_Dr1_Lft_Leaf_Clng LENGTH->2 STARTBIT :12"}
GVL.IIVD.S_Dr1_Lft_Leaf_Clng.v			:= NOT GVL.IIVD.S_TmOut_Kapi_Durum_1_0X235 AND NOT _FB_CanRx_Message_Unpack_235.S_Bit_13;
GVL.IIVD.S_Dr1_Lft_Leaf_Clng.x			:= GVL.IIVD.S_Dr1_Lft_Leaf_Clng.v AND _FB_CanRx_Message_Unpack_235.S_Bit_12;
GVL.IIVD.S_Dr1_Lft_Leaf_Clng.e			:= _FB_CanRx_Message_Unpack_235.S_Bit_13 AND NOT _FB_CanRx_Message_Unpack_235.S_Bit_12 ;
GVL.IIVD.S_Dr1_Lft_Leaf_Clng.na			:= _FB_CanRx_Message_Unpack_235.S_Bit_13 AND _FB_CanRx_Message_Unpack_235.S_Bit_12 ;
{endregion}
{region " SIGNAL AREA : NAME->S_Dr1_Lft_Leaf_Op LENGTH->2 STARTBIT :14"}
GVL.IIVD.S_Dr1_Lft_Leaf_Op.v			:= NOT GVL.IIVD.S_TmOut_Kapi_Durum_1_0X235 AND NOT _FB_CanRx_Message_Unpack_235.S_Bit_15;
GVL.IIVD.S_Dr1_Lft_Leaf_Op.x			:= GVL.IIVD.S_Dr1_Lft_Leaf_Op.v AND _FB_CanRx_Message_Unpack_235.S_Bit_14;
GVL.IIVD.S_Dr1_Lft_Leaf_Op.e			:= _FB_CanRx_Message_Unpack_235.S_Bit_15 AND NOT _FB_CanRx_Message_Unpack_235.S_Bit_14 ;
GVL.IIVD.S_Dr1_Lft_Leaf_Op.na			:= _FB_CanRx_Message_Unpack_235.S_Bit_15 AND _FB_CanRx_Message_Unpack_235.S_Bit_14 ;
{endregion}
{region " SIGNAL AREA : NAME->S_Dr1_Lft_Leaf_Cl LENGTH->2 STARTBIT :16"}
GVL.IIVD.S_Dr1_Lft_Leaf_Cl.v			:= NOT GVL.IIVD.S_TmOut_Kapi_Durum_1_0X235 AND NOT _FB_CanRx_Message_Unpack_235.S_Bit_17;
GVL.IIVD.S_Dr1_Lft_Leaf_Cl.x			:= GVL.IIVD.S_Dr1_Lft_Leaf_Cl.v AND _FB_CanRx_Message_Unpack_235.S_Bit_16;
GVL.IIVD.S_Dr1_Lft_Leaf_Cl.e			:= _FB_CanRx_Message_Unpack_235.S_Bit_17 AND NOT _FB_CanRx_Message_Unpack_235.S_Bit_16 ;
GVL.IIVD.S_Dr1_Lft_Leaf_Cl.na			:= _FB_CanRx_Message_Unpack_235.S_Bit_17 AND _FB_CanRx_Message_Unpack_235.S_Bit_16 ;
{endregion}
{region " SIGNAL AREA : NAME->S_Dr1_Lft_Leaf_Obs LENGTH->2 STARTBIT :18"}
GVL.IIVD.S_Dr1_Lft_Leaf_Obs.v			:= NOT GVL.IIVD.S_TmOut_Kapi_Durum_1_0X235 AND NOT _FB_CanRx_Message_Unpack_235.S_Bit_19;
GVL.IIVD.S_Dr1_Lft_Leaf_Obs.x			:= GVL.IIVD.S_Dr1_Lft_Leaf_Obs.v AND _FB_CanRx_Message_Unpack_235.S_Bit_18;
GVL.IIVD.S_Dr1_Lft_Leaf_Obs.e			:= _FB_CanRx_Message_Unpack_235.S_Bit_19 AND NOT _FB_CanRx_Message_Unpack_235.S_Bit_18 ;
GVL.IIVD.S_Dr1_Lft_Leaf_Obs.na			:= _FB_CanRx_Message_Unpack_235.S_Bit_19 AND _FB_CanRx_Message_Unpack_235.S_Bit_18 ;
{endregion}
{region " SIGNAL AREA : NAME->S_Dr1_Em_Swc LENGTH->2 STARTBIT :20"}
GVL.IIVD.S_Dr1_Em_Swc.v					:= NOT GVL.IIVD.S_TmOut_Kapi_Durum_1_0X235 AND NOT _FB_CanRx_Message_Unpack_235.S_Bit_21;
GVL.IIVD.S_Dr1_Em_Swc.x					:= GVL.IIVD.S_Dr1_Em_Swc.v AND _FB_CanRx_Message_Unpack_235.S_Bit_20;
GVL.IIVD.S_Dr1_Em_Swc.e					:= _FB_CanRx_Message_Unpack_235.S_Bit_21 AND NOT _FB_CanRx_Message_Unpack_235.S_Bit_20 ;
GVL.IIVD.S_Dr1_Em_Swc.na				:= _FB_CanRx_Message_Unpack_235.S_Bit_21 AND _FB_CanRx_Message_Unpack_235.S_Bit_20 ;
{endregion}
{region " SIGNAL AREA : NAME->S_Dr2_Opng LENGTH->2 STARTBIT :24"}
GVL.IIVD.S_Dr2_Opng.v					:= NOT GVL.IIVD.S_TmOut_Kapi_Durum_1_0X235 AND NOT _FB_CanRx_Message_Unpack_235.S_Bit_25;
GVL.IIVD.S_Dr2_Opng.x					:= GVL.IIVD.S_Dr2_Opng.v AND _FB_CanRx_Message_Unpack_235.S_Bit_24;
GVL.IIVD.S_Dr2_Opng.e					:= _FB_CanRx_Message_Unpack_235.S_Bit_25 AND NOT _FB_CanRx_Message_Unpack_235.S_Bit_24 ;
GVL.IIVD.S_Dr2_Opng.na					:= _FB_CanRx_Message_Unpack_235.S_Bit_25 AND _FB_CanRx_Message_Unpack_235.S_Bit_24 ;
{endregion}
{region " SIGNAL AREA : NAME->S_Dr2_Clng LENGTH->2 STARTBIT :26"}
GVL.IIVD.S_Dr2_Clng.v					:= NOT GVL.IIVD.S_TmOut_Kapi_Durum_1_0X235 AND NOT _FB_CanRx_Message_Unpack_235.S_Bit_27;
GVL.IIVD.S_Dr2_Clng.x					:= GVL.IIVD.S_Dr2_Clng.v AND _FB_CanRx_Message_Unpack_235.S_Bit_26;
GVL.IIVD.S_Dr2_Clng.e					:= _FB_CanRx_Message_Unpack_235.S_Bit_27 AND NOT _FB_CanRx_Message_Unpack_235.S_Bit_26 ;
GVL.IIVD.S_Dr2_Clng.na					:= _FB_CanRx_Message_Unpack_235.S_Bit_27 AND _FB_CanRx_Message_Unpack_235.S_Bit_26 ;
{endregion}
{region " SIGNAL AREA : NAME->S_Dr2_Op LENGTH->2 STARTBIT :28"}
GVL.IIVD.S_Dr2_Op.v						:= NOT GVL.IIVD.S_TmOut_Kapi_Durum_1_0X235 AND NOT _FB_CanRx_Message_Unpack_235.S_Bit_29;
GVL.IIVD.S_Dr2_Op.x						:= GVL.IIVD.S_Dr2_Op.v AND _FB_CanRx_Message_Unpack_235.S_Bit_28;
GVL.IIVD.S_Dr2_Op.e						:= _FB_CanRx_Message_Unpack_235.S_Bit_29 AND NOT _FB_CanRx_Message_Unpack_235.S_Bit_28 ;
GVL.IIVD.S_Dr2_Op.na					:= _FB_CanRx_Message_Unpack_235.S_Bit_29 AND _FB_CanRx_Message_Unpack_235.S_Bit_28 ;
{endregion}
{region " SIGNAL AREA : NAME->S_Dr2_Cl LENGTH->2 STARTBIT :30"}
GVL.IIVD.S_Dr2_Cl.v						:= NOT GVL.IIVD.S_TmOut_Kapi_Durum_1_0X235 AND NOT _FB_CanRx_Message_Unpack_235.S_Bit_31;
GVL.IIVD.S_Dr2_Cl.x						:= GVL.IIVD.S_Dr2_Cl.v AND _FB_CanRx_Message_Unpack_235.S_Bit_30;
GVL.IIVD.S_Dr2_Cl.e						:= _FB_CanRx_Message_Unpack_235.S_Bit_31 AND NOT _FB_CanRx_Message_Unpack_235.S_Bit_30 ;
GVL.IIVD.S_Dr2_Cl.na					:= _FB_CanRx_Message_Unpack_235.S_Bit_31 AND _FB_CanRx_Message_Unpack_235.S_Bit_30 ;
{endregion}
{region " SIGNAL AREA : NAME->S_Dr2_Obs LENGTH->2 STARTBIT :32"}
GVL.IIVD.S_Dr2_Obs.v					:= NOT GVL.IIVD.S_TmOut_Kapi_Durum_1_0X235 AND NOT _FB_CanRx_Message_Unpack_235.S_Bit_33;
GVL.IIVD.S_Dr2_Obs.x					:= GVL.IIVD.S_Dr2_Obs.v AND _FB_CanRx_Message_Unpack_235.S_Bit_32;
GVL.IIVD.S_Dr2_Obs.e					:= _FB_CanRx_Message_Unpack_235.S_Bit_33 AND NOT _FB_CanRx_Message_Unpack_235.S_Bit_32 ;
GVL.IIVD.S_Dr2_Obs.na					:= _FB_CanRx_Message_Unpack_235.S_Bit_33 AND _FB_CanRx_Message_Unpack_235.S_Bit_32 ;
{endregion}
{region " SIGNAL AREA : NAME->S_Dr2_Em_Swc LENGTH->2 STARTBIT :34"}
GVL.IIVD.S_Dr2_Em_Swc.v					:= NOT GVL.IIVD.S_TmOut_Kapi_Durum_1_0X235 AND NOT _FB_CanRx_Message_Unpack_235.S_Bit_35;
GVL.IIVD.S_Dr2_Em_Swc.x					:= GVL.IIVD.S_Dr2_Em_Swc.v AND _FB_CanRx_Message_Unpack_235.S_Bit_34;
GVL.IIVD.S_Dr2_Em_Swc.e					:= _FB_CanRx_Message_Unpack_235.S_Bit_35 AND NOT _FB_CanRx_Message_Unpack_235.S_Bit_34 ;
GVL.IIVD.S_Dr2_Em_Swc.na				:= _FB_CanRx_Message_Unpack_235.S_Bit_35 AND _FB_CanRx_Message_Unpack_235.S_Bit_34 ;
{endregion}
{region " SIGNAL AREA : NAME->S_Dr3_Opng LENGTH->2 STARTBIT :40"}
GVL.IIVD.S_Dr3_Opng.v					:= NOT GVL.IIVD.S_TmOut_Kapi_Durum_1_0X235 AND NOT _FB_CanRx_Message_Unpack_235.S_Bit_41;
GVL.IIVD.S_Dr3_Opng.x					:= GVL.IIVD.S_Dr3_Opng.v AND _FB_CanRx_Message_Unpack_235.S_Bit_40;
GVL.IIVD.S_Dr3_Opng.e					:= _FB_CanRx_Message_Unpack_235.S_Bit_41 AND NOT _FB_CanRx_Message_Unpack_235.S_Bit_40 ;
GVL.IIVD.S_Dr3_Opng.na					:= _FB_CanRx_Message_Unpack_235.S_Bit_41 AND _FB_CanRx_Message_Unpack_235.S_Bit_40 ;
{endregion}
{region " SIGNAL AREA : NAME->S_Dr3_Clng LENGTH->2 STARTBIT :42"}
GVL.IIVD.S_Dr3_Clng.v					:= NOT GVL.IIVD.S_TmOut_Kapi_Durum_1_0X235 AND NOT _FB_CanRx_Message_Unpack_235.S_Bit_43;
GVL.IIVD.S_Dr3_Clng.x					:= GVL.IIVD.S_Dr3_Clng.v AND _FB_CanRx_Message_Unpack_235.S_Bit_42;
GVL.IIVD.S_Dr3_Clng.e					:= _FB_CanRx_Message_Unpack_235.S_Bit_43 AND NOT _FB_CanRx_Message_Unpack_235.S_Bit_42 ;
GVL.IIVD.S_Dr3_Clng.na					:= _FB_CanRx_Message_Unpack_235.S_Bit_43 AND _FB_CanRx_Message_Unpack_235.S_Bit_42 ;
{endregion}
{region " SIGNAL AREA : NAME->S_Dr3_Op LENGTH->2 STARTBIT :44"}
GVL.IIVD.S_Dr3_Op.v						:= NOT GVL.IIVD.S_TmOut_Kapi_Durum_1_0X235 AND NOT _FB_CanRx_Message_Unpack_235.S_Bit_45;
GVL.IIVD.S_Dr3_Op.x						:= GVL.IIVD.S_Dr3_Op.v AND _FB_CanRx_Message_Unpack_235.S_Bit_44;
GVL.IIVD.S_Dr3_Op.e						:= _FB_CanRx_Message_Unpack_235.S_Bit_45 AND NOT _FB_CanRx_Message_Unpack_235.S_Bit_44 ;
GVL.IIVD.S_Dr3_Op.na					:= _FB_CanRx_Message_Unpack_235.S_Bit_45 AND _FB_CanRx_Message_Unpack_235.S_Bit_44 ;
{endregion}
{region " SIGNAL AREA : NAME->S_Dr3_Cl LENGTH->2 STARTBIT :46"}
GVL.IIVD.S_Dr3_Cl.v						:= NOT GVL.IIVD.S_TmOut_Kapi_Durum_1_0X235 AND NOT _FB_CanRx_Message_Unpack_235.S_Bit_47;
GVL.IIVD.S_Dr3_Cl.x						:= GVL.IIVD.S_Dr3_Cl.v AND _FB_CanRx_Message_Unpack_235.S_Bit_46;
GVL.IIVD.S_Dr3_Cl.e						:= _FB_CanRx_Message_Unpack_235.S_Bit_47 AND NOT _FB_CanRx_Message_Unpack_235.S_Bit_46 ;
GVL.IIVD.S_Dr3_Cl.na					:= _FB_CanRx_Message_Unpack_235.S_Bit_47 AND _FB_CanRx_Message_Unpack_235.S_Bit_46 ;
{endregion}
{region " SIGNAL AREA : NAME->S_Dr3_Obs LENGTH->2 STARTBIT :48"}
GVL.IIVD.S_Dr3_Obs.v					:= NOT GVL.IIVD.S_TmOut_Kapi_Durum_1_0X235 AND NOT _FB_CanRx_Message_Unpack_235.S_Bit_49;
GVL.IIVD.S_Dr3_Obs.x					:= GVL.IIVD.S_Dr3_Obs.v AND _FB_CanRx_Message_Unpack_235.S_Bit_48;
GVL.IIVD.S_Dr3_Obs.e					:= _FB_CanRx_Message_Unpack_235.S_Bit_49 AND NOT _FB_CanRx_Message_Unpack_235.S_Bit_48 ;
GVL.IIVD.S_Dr3_Obs.na					:= _FB_CanRx_Message_Unpack_235.S_Bit_49 AND _FB_CanRx_Message_Unpack_235.S_Bit_48 ;
{endregion}
{region " SIGNAL AREA : NAME->S_Dr3_Em_Swc LENGTH->2 STARTBIT :50"}
GVL.IIVD.S_Dr3_Em_Swc.v					:= NOT GVL.IIVD.S_TmOut_Kapi_Durum_1_0X235 AND NOT _FB_CanRx_Message_Unpack_235.S_Bit_51;
GVL.IIVD.S_Dr3_Em_Swc.x					:= GVL.IIVD.S_Dr3_Em_Swc.v AND _FB_CanRx_Message_Unpack_235.S_Bit_50;
GVL.IIVD.S_Dr3_Em_Swc.e					:= _FB_CanRx_Message_Unpack_235.S_Bit_51 AND NOT _FB_CanRx_Message_Unpack_235.S_Bit_50 ;
GVL.IIVD.S_Dr3_Em_Swc.na				:= _FB_CanRx_Message_Unpack_235.S_Bit_51 AND _FB_CanRx_Message_Unpack_235.S_Bit_50 ;
{endregion}
{endregion}

{region " MESSAGE AREA :Kapi_Durum_2- ID:237"}

_FB_CanRx_Message_Unpack_237 (		C_Enable	:= GVL.IIVD.S_CAN_Init,
     								Obj_CAN		:= ADR(GVL.IC.Obj_CAN0),
     								X_MsgID		:= 16#237,
     								Tm_MsgTmOut	:= TIME#2500MS,
     								S_Extended	:= 0,
     								S_ER_TmOut	=> GVL.IIVD.S_TmOut_Kapi_Durum_2_0X237);

{region " SIGNAL AREA : NAME->S_Dr4_Opng LENGTH->2 STARTBIT :0"}
GVL.IIVD.S_Dr4_Opng.v					:= NOT GVL.IIVD.S_TmOut_Kapi_Durum_2_0X237 AND NOT _FB_CanRx_Message_Unpack_237.S_Bit_1;
GVL.IIVD.S_Dr4_Opng.x					:= GVL.IIVD.S_Dr4_Opng.v AND _FB_CanRx_Message_Unpack_237.S_Bit_0;
GVL.IIVD.S_Dr4_Opng.e					:= _FB_CanRx_Message_Unpack_237.S_Bit_1 AND NOT _FB_CanRx_Message_Unpack_237.S_Bit_0 ;
GVL.IIVD.S_Dr4_Opng.na					:= _FB_CanRx_Message_Unpack_237.S_Bit_1 AND _FB_CanRx_Message_Unpack_237.S_Bit_0 ;
{endregion}
{region " SIGNAL AREA : NAME->S_Dr4_Clng LENGTH->2 STARTBIT :2"}
GVL.IIVD.S_Dr4_Clng.v					:= NOT GVL.IIVD.S_TmOut_Kapi_Durum_2_0X237 AND NOT _FB_CanRx_Message_Unpack_237.S_Bit_3;
GVL.IIVD.S_Dr4_Clng.x					:= GVL.IIVD.S_Dr4_Clng.v AND _FB_CanRx_Message_Unpack_237.S_Bit_2;
GVL.IIVD.S_Dr4_Clng.e					:= _FB_CanRx_Message_Unpack_237.S_Bit_3 AND NOT _FB_CanRx_Message_Unpack_237.S_Bit_2 ;
GVL.IIVD.S_Dr4_Clng.na					:= _FB_CanRx_Message_Unpack_237.S_Bit_3 AND _FB_CanRx_Message_Unpack_237.S_Bit_2 ;
{endregion}
{region " SIGNAL AREA : NAME->S_Dr4_Op LENGTH->2 STARTBIT :4"}
GVL.IIVD.S_Dr4_Op.v						:= NOT GVL.IIVD.S_TmOut_Kapi_Durum_2_0X237 AND NOT _FB_CanRx_Message_Unpack_237.S_Bit_5;
GVL.IIVD.S_Dr4_Op.x						:= GVL.IIVD.S_Dr4_Op.v AND _FB_CanRx_Message_Unpack_237.S_Bit_4;
GVL.IIVD.S_Dr4_Op.e						:= _FB_CanRx_Message_Unpack_237.S_Bit_5 AND NOT _FB_CanRx_Message_Unpack_237.S_Bit_4 ;
GVL.IIVD.S_Dr4_Op.na					:= _FB_CanRx_Message_Unpack_237.S_Bit_5 AND _FB_CanRx_Message_Unpack_237.S_Bit_4 ;
{endregion}
{region " SIGNAL AREA : NAME->S_Dr4_Cl LENGTH->2 STARTBIT :6"}
GVL.IIVD.S_Dr4_Cl.v						:= NOT GVL.IIVD.S_TmOut_Kapi_Durum_2_0X237 AND NOT _FB_CanRx_Message_Unpack_237.S_Bit_7;
GVL.IIVD.S_Dr4_Cl.x						:= GVL.IIVD.S_Dr4_Cl.v AND _FB_CanRx_Message_Unpack_237.S_Bit_6;
GVL.IIVD.S_Dr4_Cl.e						:= _FB_CanRx_Message_Unpack_237.S_Bit_7 AND NOT _FB_CanRx_Message_Unpack_237.S_Bit_6 ;
GVL.IIVD.S_Dr4_Cl.na					:= _FB_CanRx_Message_Unpack_237.S_Bit_7 AND _FB_CanRx_Message_Unpack_237.S_Bit_6 ;
{endregion}
{region " SIGNAL AREA : NAME->S_Dr4_Obs LENGTH->2 STARTBIT :8"}
GVL.IIVD.S_Dr4_Obs.v					:= NOT GVL.IIVD.S_TmOut_Kapi_Durum_2_0X237 AND NOT _FB_CanRx_Message_Unpack_237.S_Bit_9;
GVL.IIVD.S_Dr4_Obs.x					:= GVL.IIVD.S_Dr4_Obs.v AND _FB_CanRx_Message_Unpack_237.S_Bit_8;
GVL.IIVD.S_Dr4_Obs.e					:= _FB_CanRx_Message_Unpack_237.S_Bit_9 AND NOT _FB_CanRx_Message_Unpack_237.S_Bit_8 ;
GVL.IIVD.S_Dr4_Obs.na					:= _FB_CanRx_Message_Unpack_237.S_Bit_9 AND _FB_CanRx_Message_Unpack_237.S_Bit_8 ;
{endregion}
{region " SIGNAL AREA : NAME->S_Dr4_Em_Swc LENGTH->2 STARTBIT :10"}
GVL.IIVD.S_Dr4_Em_Swc.v					:= NOT GVL.IIVD.S_TmOut_Kapi_Durum_2_0X237 AND NOT _FB_CanRx_Message_Unpack_237.S_Bit_11;
GVL.IIVD.S_Dr4_Em_Swc.x					:= GVL.IIVD.S_Dr4_Em_Swc.v AND _FB_CanRx_Message_Unpack_237.S_Bit_10;
GVL.IIVD.S_Dr4_Em_Swc.e					:= _FB_CanRx_Message_Unpack_237.S_Bit_11 AND NOT _FB_CanRx_Message_Unpack_237.S_Bit_10 ;
GVL.IIVD.S_Dr4_Em_Swc.na				:= _FB_CanRx_Message_Unpack_237.S_Bit_11 AND _FB_CanRx_Message_Unpack_237.S_Bit_10 ;
{endregion}
{region " SIGNAL AREA : NAME->S_Dr5_Opng LENGTH->2 STARTBIT :16"}
GVL.IIVD.S_Dr5_Opng.v					:= NOT GVL.IIVD.S_TmOut_Kapi_Durum_2_0X237 AND NOT _FB_CanRx_Message_Unpack_237.S_Bit_17;
GVL.IIVD.S_Dr5_Opng.x					:= GVL.IIVD.S_Dr5_Opng.v AND _FB_CanRx_Message_Unpack_237.S_Bit_16;
GVL.IIVD.S_Dr5_Opng.e					:= _FB_CanRx_Message_Unpack_237.S_Bit_17 AND NOT _FB_CanRx_Message_Unpack_237.S_Bit_16 ;
GVL.IIVD.S_Dr5_Opng.na					:= _FB_CanRx_Message_Unpack_237.S_Bit_17 AND _FB_CanRx_Message_Unpack_237.S_Bit_16 ;
{endregion}
{region " SIGNAL AREA : NAME->S_Dr5_Clng LENGTH->2 STARTBIT :18"}
GVL.IIVD.S_Dr5_Clng.v					:= NOT GVL.IIVD.S_TmOut_Kapi_Durum_2_0X237 AND NOT _FB_CanRx_Message_Unpack_237.S_Bit_19;
GVL.IIVD.S_Dr5_Clng.x					:= GVL.IIVD.S_Dr5_Clng.v AND _FB_CanRx_Message_Unpack_237.S_Bit_18;
GVL.IIVD.S_Dr5_Clng.e					:= _FB_CanRx_Message_Unpack_237.S_Bit_19 AND NOT _FB_CanRx_Message_Unpack_237.S_Bit_18 ;
GVL.IIVD.S_Dr5_Clng.na					:= _FB_CanRx_Message_Unpack_237.S_Bit_19 AND _FB_CanRx_Message_Unpack_237.S_Bit_18 ;
{endregion}
{region " SIGNAL AREA : NAME->S_Dr5_Op LENGTH->2 STARTBIT :20"}
GVL.IIVD.S_Dr5_Op.v						:= NOT GVL.IIVD.S_TmOut_Kapi_Durum_2_0X237 AND NOT _FB_CanRx_Message_Unpack_237.S_Bit_21;
GVL.IIVD.S_Dr5_Op.x						:= GVL.IIVD.S_Dr5_Op.v AND _FB_CanRx_Message_Unpack_237.S_Bit_20;
GVL.IIVD.S_Dr5_Op.e						:= _FB_CanRx_Message_Unpack_237.S_Bit_21 AND NOT _FB_CanRx_Message_Unpack_237.S_Bit_20 ;
GVL.IIVD.S_Dr5_Op.na					:= _FB_CanRx_Message_Unpack_237.S_Bit_21 AND _FB_CanRx_Message_Unpack_237.S_Bit_20 ;
{endregion}
{region " SIGNAL AREA : NAME->S_Dr5_Cl LENGTH->2 STARTBIT :22"}
GVL.IIVD.S_Dr5_Cl.v						:= NOT GVL.IIVD.S_TmOut_Kapi_Durum_2_0X237 AND NOT _FB_CanRx_Message_Unpack_237.S_Bit_23;
GVL.IIVD.S_Dr5_Cl.x						:= GVL.IIVD.S_Dr5_Cl.v AND _FB_CanRx_Message_Unpack_237.S_Bit_22;
GVL.IIVD.S_Dr5_Cl.e						:= _FB_CanRx_Message_Unpack_237.S_Bit_23 AND NOT _FB_CanRx_Message_Unpack_237.S_Bit_22 ;
GVL.IIVD.S_Dr5_Cl.na					:= _FB_CanRx_Message_Unpack_237.S_Bit_23 AND _FB_CanRx_Message_Unpack_237.S_Bit_22 ;
{endregion}
{region " SIGNAL AREA : NAME->S_Dr5_Obs LENGTH->2 STARTBIT :24"}
GVL.IIVD.S_Dr5_Obs.v					:= NOT GVL.IIVD.S_TmOut_Kapi_Durum_2_0X237 AND NOT _FB_CanRx_Message_Unpack_237.S_Bit_25;
GVL.IIVD.S_Dr5_Obs.x					:= GVL.IIVD.S_Dr5_Obs.v AND _FB_CanRx_Message_Unpack_237.S_Bit_24;
GVL.IIVD.S_Dr5_Obs.e					:= _FB_CanRx_Message_Unpack_237.S_Bit_25 AND NOT _FB_CanRx_Message_Unpack_237.S_Bit_24 ;
GVL.IIVD.S_Dr5_Obs.na					:= _FB_CanRx_Message_Unpack_237.S_Bit_25 AND _FB_CanRx_Message_Unpack_237.S_Bit_24 ;
{endregion}
{region " SIGNAL AREA : NAME->S_Dr5_Em_Swc LENGTH->2 STARTBIT :26"}
GVL.IIVD.S_Dr5_Em_Swc.v					:= NOT GVL.IIVD.S_TmOut_Kapi_Durum_2_0X237 AND NOT _FB_CanRx_Message_Unpack_237.S_Bit_27;
GVL.IIVD.S_Dr5_Em_Swc.x					:= GVL.IIVD.S_Dr5_Em_Swc.v AND _FB_CanRx_Message_Unpack_237.S_Bit_26;
GVL.IIVD.S_Dr5_Em_Swc.e					:= _FB_CanRx_Message_Unpack_237.S_Bit_27 AND NOT _FB_CanRx_Message_Unpack_237.S_Bit_26 ;
GVL.IIVD.S_Dr5_Em_Swc.na				:= _FB_CanRx_Message_Unpack_237.S_Bit_27 AND _FB_CanRx_Message_Unpack_237.S_Bit_26 ;
{endregion}
{region " SIGNAL AREA : NAME->S_Dr6_Opng LENGTH->2 STARTBIT :32"}
GVL.IIVD.S_Dr6_Opng.v					:= NOT GVL.IIVD.S_TmOut_Kapi_Durum_2_0X237 AND NOT _FB_CanRx_Message_Unpack_237.S_Bit_33;
GVL.IIVD.S_Dr6_Opng.x					:= GVL.IIVD.S_Dr6_Opng.v AND _FB_CanRx_Message_Unpack_237.S_Bit_32;
GVL.IIVD.S_Dr6_Opng.e					:= _FB_CanRx_Message_Unpack_237.S_Bit_33 AND NOT _FB_CanRx_Message_Unpack_237.S_Bit_32 ;
GVL.IIVD.S_Dr6_Opng.na					:= _FB_CanRx_Message_Unpack_237.S_Bit_33 AND _FB_CanRx_Message_Unpack_237.S_Bit_32 ;
{endregion}
{region " SIGNAL AREA : NAME->S_Dr6_Clng LENGTH->2 STARTBIT :34"}
GVL.IIVD.S_Dr6_Clng.v					:= NOT GVL.IIVD.S_TmOut_Kapi_Durum_2_0X237 AND NOT _FB_CanRx_Message_Unpack_237.S_Bit_35;
GVL.IIVD.S_Dr6_Clng.x					:= GVL.IIVD.S_Dr6_Clng.v AND _FB_CanRx_Message_Unpack_237.S_Bit_34;
GVL.IIVD.S_Dr6_Clng.e					:= _FB_CanRx_Message_Unpack_237.S_Bit_35 AND NOT _FB_CanRx_Message_Unpack_237.S_Bit_34 ;
GVL.IIVD.S_Dr6_Clng.na					:= _FB_CanRx_Message_Unpack_237.S_Bit_35 AND _FB_CanRx_Message_Unpack_237.S_Bit_34 ;
{endregion}
{region " SIGNAL AREA : NAME->S_Dr6_Op LENGTH->2 STARTBIT :36"}
GVL.IIVD.S_Dr6_Op.v						:= NOT GVL.IIVD.S_TmOut_Kapi_Durum_2_0X237 AND NOT _FB_CanRx_Message_Unpack_237.S_Bit_37;
GVL.IIVD.S_Dr6_Op.x						:= GVL.IIVD.S_Dr6_Op.v AND _FB_CanRx_Message_Unpack_237.S_Bit_36;
GVL.IIVD.S_Dr6_Op.e						:= _FB_CanRx_Message_Unpack_237.S_Bit_37 AND NOT _FB_CanRx_Message_Unpack_237.S_Bit_36 ;
GVL.IIVD.S_Dr6_Op.na					:= _FB_CanRx_Message_Unpack_237.S_Bit_37 AND _FB_CanRx_Message_Unpack_237.S_Bit_36 ;
{endregion}
{region " SIGNAL AREA : NAME->S_Dr6_Cl LENGTH->2 STARTBIT :38"}
GVL.IIVD.S_Dr6_Cl.v						:= NOT GVL.IIVD.S_TmOut_Kapi_Durum_2_0X237 AND NOT _FB_CanRx_Message_Unpack_237.S_Bit_39;
GVL.IIVD.S_Dr6_Cl.x						:= GVL.IIVD.S_Dr6_Cl.v AND _FB_CanRx_Message_Unpack_237.S_Bit_38;
GVL.IIVD.S_Dr6_Cl.e						:= _FB_CanRx_Message_Unpack_237.S_Bit_39 AND NOT _FB_CanRx_Message_Unpack_237.S_Bit_38 ;
GVL.IIVD.S_Dr6_Cl.na					:= _FB_CanRx_Message_Unpack_237.S_Bit_39 AND _FB_CanRx_Message_Unpack_237.S_Bit_38 ;
{endregion}
{region " SIGNAL AREA : NAME->S_Dr6_Obs LENGTH->2 STARTBIT :40"}
GVL.IIVD.S_Dr6_Obs.v					:= NOT GVL.IIVD.S_TmOut_Kapi_Durum_2_0X237 AND NOT _FB_CanRx_Message_Unpack_237.S_Bit_41;
GVL.IIVD.S_Dr6_Obs.x					:= GVL.IIVD.S_Dr6_Obs.v AND _FB_CanRx_Message_Unpack_237.S_Bit_40;
GVL.IIVD.S_Dr6_Obs.e					:= _FB_CanRx_Message_Unpack_237.S_Bit_41 AND NOT _FB_CanRx_Message_Unpack_237.S_Bit_40 ;
GVL.IIVD.S_Dr6_Obs.na					:= _FB_CanRx_Message_Unpack_237.S_Bit_41 AND _FB_CanRx_Message_Unpack_237.S_Bit_40 ;
{endregion}
{region " SIGNAL AREA : NAME->S_Dr6_Em_Swc LENGTH->2 STARTBIT :42"}
GVL.IIVD.S_Dr6_Em_Swc.v					:= NOT GVL.IIVD.S_TmOut_Kapi_Durum_2_0X237 AND NOT _FB_CanRx_Message_Unpack_237.S_Bit_43;
GVL.IIVD.S_Dr6_Em_Swc.x					:= GVL.IIVD.S_Dr6_Em_Swc.v AND _FB_CanRx_Message_Unpack_237.S_Bit_42;
GVL.IIVD.S_Dr6_Em_Swc.e					:= _FB_CanRx_Message_Unpack_237.S_Bit_43 AND NOT _FB_CanRx_Message_Unpack_237.S_Bit_42 ;
GVL.IIVD.S_Dr6_Em_Swc.na				:= _FB_CanRx_Message_Unpack_237.S_Bit_43 AND _FB_CanRx_Message_Unpack_237.S_Bit_42 ;
{endregion}
{endregion}

{region " MESSAGE AREA :Kapi_Durum_3- ID:238"}

_FB_CanRx_Message_Unpack_238 (		C_Enable	:= GVL.IIVD.S_CAN_Init,
     								Obj_CAN		:= ADR(GVL.IC.Obj_CAN0),
     								X_MsgID		:= 16#238,
     								Tm_MsgTmOut	:= TIME#2500MS,
     								S_Extended	:= 0,
     								S_ER_TmOut	=> GVL.IIVD.S_TmOut_Kapi_Durum_3_0X238);

{region " SIGNAL AREA : NAME->S_Dr7_Opng LENGTH->2 STARTBIT :0"}
GVL.IIVD.S_Dr7_Opng.v					:= NOT GVL.IIVD.S_TmOut_Kapi_Durum_3_0X238 AND NOT _FB_CanRx_Message_Unpack_238.S_Bit_1;
GVL.IIVD.S_Dr7_Opng.x					:= GVL.IIVD.S_Dr7_Opng.v AND _FB_CanRx_Message_Unpack_238.S_Bit_0;
GVL.IIVD.S_Dr7_Opng.e					:= _FB_CanRx_Message_Unpack_238.S_Bit_1 AND NOT _FB_CanRx_Message_Unpack_238.S_Bit_0 ;
GVL.IIVD.S_Dr7_Opng.na					:= _FB_CanRx_Message_Unpack_238.S_Bit_1 AND _FB_CanRx_Message_Unpack_238.S_Bit_0 ;
{endregion}
{region " SIGNAL AREA : NAME->S_Dr7_Clng LENGTH->2 STARTBIT :2"}
GVL.IIVD.S_Dr7_Clng.v					:= NOT GVL.IIVD.S_TmOut_Kapi_Durum_3_0X238 AND NOT _FB_CanRx_Message_Unpack_238.S_Bit_3;
GVL.IIVD.S_Dr7_Clng.x					:= GVL.IIVD.S_Dr7_Clng.v AND _FB_CanRx_Message_Unpack_238.S_Bit_2;
GVL.IIVD.S_Dr7_Clng.e					:= _FB_CanRx_Message_Unpack_238.S_Bit_3 AND NOT _FB_CanRx_Message_Unpack_238.S_Bit_2 ;
GVL.IIVD.S_Dr7_Clng.na					:= _FB_CanRx_Message_Unpack_238.S_Bit_3 AND _FB_CanRx_Message_Unpack_238.S_Bit_2 ;
{endregion}
{region " SIGNAL AREA : NAME->S_Dr7_Op LENGTH->2 STARTBIT :4"}
GVL.IIVD.S_Dr7_Op.v						:= NOT GVL.IIVD.S_TmOut_Kapi_Durum_3_0X238 AND NOT _FB_CanRx_Message_Unpack_238.S_Bit_5;
GVL.IIVD.S_Dr7_Op.x						:= GVL.IIVD.S_Dr7_Op.v AND _FB_CanRx_Message_Unpack_238.S_Bit_4;
GVL.IIVD.S_Dr7_Op.e						:= _FB_CanRx_Message_Unpack_238.S_Bit_5 AND NOT _FB_CanRx_Message_Unpack_238.S_Bit_4 ;
GVL.IIVD.S_Dr7_Op.na					:= _FB_CanRx_Message_Unpack_238.S_Bit_5 AND _FB_CanRx_Message_Unpack_238.S_Bit_4 ;
{endregion}
{region " SIGNAL AREA : NAME->S_Dr7_Cl LENGTH->2 STARTBIT :6"}
GVL.IIVD.S_Dr7_Cl.v						:= NOT GVL.IIVD.S_TmOut_Kapi_Durum_3_0X238 AND NOT _FB_CanRx_Message_Unpack_238.S_Bit_7;
GVL.IIVD.S_Dr7_Cl.x						:= GVL.IIVD.S_Dr7_Cl.v AND _FB_CanRx_Message_Unpack_238.S_Bit_6;
GVL.IIVD.S_Dr7_Cl.e						:= _FB_CanRx_Message_Unpack_238.S_Bit_7 AND NOT _FB_CanRx_Message_Unpack_238.S_Bit_6 ;
GVL.IIVD.S_Dr7_Cl.na					:= _FB_CanRx_Message_Unpack_238.S_Bit_7 AND _FB_CanRx_Message_Unpack_238.S_Bit_6 ;
{endregion}
{region " SIGNAL AREA : NAME->S_Dr7_Obs LENGTH->2 STARTBIT :8"}
GVL.IIVD.S_Dr7_Obs.v					:= NOT GVL.IIVD.S_TmOut_Kapi_Durum_3_0X238 AND NOT _FB_CanRx_Message_Unpack_238.S_Bit_9;
GVL.IIVD.S_Dr7_Obs.x					:= GVL.IIVD.S_Dr7_Obs.v AND _FB_CanRx_Message_Unpack_238.S_Bit_8;
GVL.IIVD.S_Dr7_Obs.e					:= _FB_CanRx_Message_Unpack_238.S_Bit_9 AND NOT _FB_CanRx_Message_Unpack_238.S_Bit_8 ;
GVL.IIVD.S_Dr7_Obs.na					:= _FB_CanRx_Message_Unpack_238.S_Bit_9 AND _FB_CanRx_Message_Unpack_238.S_Bit_8 ;
{endregion}
{region " SIGNAL AREA : NAME->S_Dr7_Em_Swc LENGTH->2 STARTBIT :10"}
GVL.IIVD.S_Dr7_Em_Swc.v					:= NOT GVL.IIVD.S_TmOut_Kapi_Durum_3_0X238 AND NOT _FB_CanRx_Message_Unpack_238.S_Bit_11;
GVL.IIVD.S_Dr7_Em_Swc.x					:= GVL.IIVD.S_Dr7_Em_Swc.v AND _FB_CanRx_Message_Unpack_238.S_Bit_10;
GVL.IIVD.S_Dr7_Em_Swc.e					:= _FB_CanRx_Message_Unpack_238.S_Bit_11 AND NOT _FB_CanRx_Message_Unpack_238.S_Bit_10 ;
GVL.IIVD.S_Dr7_Em_Swc.na				:= _FB_CanRx_Message_Unpack_238.S_Bit_11 AND _FB_CanRx_Message_Unpack_238.S_Bit_10 ;
{endregion}
{region " SIGNAL AREA : NAME->S_Dr8_Opng LENGTH->2 STARTBIT :16"}
GVL.IIVD.S_Dr8_Opng.v					:= NOT GVL.IIVD.S_TmOut_Kapi_Durum_3_0X238 AND NOT _FB_CanRx_Message_Unpack_238.S_Bit_17;
GVL.IIVD.S_Dr8_Opng.x					:= GVL.IIVD.S_Dr8_Opng.v AND _FB_CanRx_Message_Unpack_238.S_Bit_16;
GVL.IIVD.S_Dr8_Opng.e					:= _FB_CanRx_Message_Unpack_238.S_Bit_17 AND NOT _FB_CanRx_Message_Unpack_238.S_Bit_16 ;
GVL.IIVD.S_Dr8_Opng.na					:= _FB_CanRx_Message_Unpack_238.S_Bit_17 AND _FB_CanRx_Message_Unpack_238.S_Bit_16 ;
{endregion}
{region " SIGNAL AREA : NAME->S_Dr8_Clng LENGTH->2 STARTBIT :18"}
GVL.IIVD.S_Dr8_Clng.v					:= NOT GVL.IIVD.S_TmOut_Kapi_Durum_3_0X238 AND NOT _FB_CanRx_Message_Unpack_238.S_Bit_19;
GVL.IIVD.S_Dr8_Clng.x					:= GVL.IIVD.S_Dr8_Clng.v AND _FB_CanRx_Message_Unpack_238.S_Bit_18;
GVL.IIVD.S_Dr8_Clng.e					:= _FB_CanRx_Message_Unpack_238.S_Bit_19 AND NOT _FB_CanRx_Message_Unpack_238.S_Bit_18 ;
GVL.IIVD.S_Dr8_Clng.na					:= _FB_CanRx_Message_Unpack_238.S_Bit_19 AND _FB_CanRx_Message_Unpack_238.S_Bit_18 ;
{endregion}
{region " SIGNAL AREA : NAME->S_Dr8_Op LENGTH->2 STARTBIT :20"}
GVL.IIVD.S_Dr8_Op.v						:= NOT GVL.IIVD.S_TmOut_Kapi_Durum_3_0X238 AND NOT _FB_CanRx_Message_Unpack_238.S_Bit_21;
GVL.IIVD.S_Dr8_Op.x						:= GVL.IIVD.S_Dr8_Op.v AND _FB_CanRx_Message_Unpack_238.S_Bit_20;
GVL.IIVD.S_Dr8_Op.e						:= _FB_CanRx_Message_Unpack_238.S_Bit_21 AND NOT _FB_CanRx_Message_Unpack_238.S_Bit_20 ;
GVL.IIVD.S_Dr8_Op.na					:= _FB_CanRx_Message_Unpack_238.S_Bit_21 AND _FB_CanRx_Message_Unpack_238.S_Bit_20 ;
{endregion}
{region " SIGNAL AREA : NAME->S_Dr8_Cl LENGTH->2 STARTBIT :22"}
GVL.IIVD.S_Dr8_Cl.v						:= NOT GVL.IIVD.S_TmOut_Kapi_Durum_3_0X238 AND NOT _FB_CanRx_Message_Unpack_238.S_Bit_23;
GVL.IIVD.S_Dr8_Cl.x						:= GVL.IIVD.S_Dr8_Cl.v AND _FB_CanRx_Message_Unpack_238.S_Bit_22;
GVL.IIVD.S_Dr8_Cl.e						:= _FB_CanRx_Message_Unpack_238.S_Bit_23 AND NOT _FB_CanRx_Message_Unpack_238.S_Bit_22 ;
GVL.IIVD.S_Dr8_Cl.na					:= _FB_CanRx_Message_Unpack_238.S_Bit_23 AND _FB_CanRx_Message_Unpack_238.S_Bit_22 ;
{endregion}
{region " SIGNAL AREA : NAME->S_Dr8_Obs LENGTH->2 STARTBIT :24"}
GVL.IIVD.S_Dr8_Obs.v					:= NOT GVL.IIVD.S_TmOut_Kapi_Durum_3_0X238 AND NOT _FB_CanRx_Message_Unpack_238.S_Bit_25;
GVL.IIVD.S_Dr8_Obs.x					:= GVL.IIVD.S_Dr8_Obs.v AND _FB_CanRx_Message_Unpack_238.S_Bit_24;
GVL.IIVD.S_Dr8_Obs.e					:= _FB_CanRx_Message_Unpack_238.S_Bit_25 AND NOT _FB_CanRx_Message_Unpack_238.S_Bit_24 ;
GVL.IIVD.S_Dr8_Obs.na					:= _FB_CanRx_Message_Unpack_238.S_Bit_25 AND _FB_CanRx_Message_Unpack_238.S_Bit_24 ;
{endregion}
{region " SIGNAL AREA : NAME->S_Dr8_Em_Swc LENGTH->2 STARTBIT :26"}
GVL.IIVD.S_Dr8_Em_Swc.v					:= NOT GVL.IIVD.S_TmOut_Kapi_Durum_3_0X238 AND NOT _FB_CanRx_Message_Unpack_238.S_Bit_27;
GVL.IIVD.S_Dr8_Em_Swc.x					:= GVL.IIVD.S_Dr8_Em_Swc.v AND _FB_CanRx_Message_Unpack_238.S_Bit_26;
GVL.IIVD.S_Dr8_Em_Swc.e					:= _FB_CanRx_Message_Unpack_238.S_Bit_27 AND NOT _FB_CanRx_Message_Unpack_238.S_Bit_26 ;
GVL.IIVD.S_Dr8_Em_Swc.na				:= _FB_CanRx_Message_Unpack_238.S_Bit_27 AND _FB_CanRx_Message_Unpack_238.S_Bit_26 ;
{endregion}
{region " SIGNAL AREA : NAME->S_Dr9_Opng LENGTH->2 STARTBIT :32"}
GVL.IIVD.S_Dr9_Opng.v					:= NOT GVL.IIVD.S_TmOut_Kapi_Durum_3_0X238 AND NOT _FB_CanRx_Message_Unpack_238.S_Bit_33;
GVL.IIVD.S_Dr9_Opng.x					:= GVL.IIVD.S_Dr9_Opng.v AND _FB_CanRx_Message_Unpack_238.S_Bit_32;
GVL.IIVD.S_Dr9_Opng.e					:= _FB_CanRx_Message_Unpack_238.S_Bit_33 AND NOT _FB_CanRx_Message_Unpack_238.S_Bit_32 ;
GVL.IIVD.S_Dr9_Opng.na					:= _FB_CanRx_Message_Unpack_238.S_Bit_33 AND _FB_CanRx_Message_Unpack_238.S_Bit_32 ;
{endregion}
{region " SIGNAL AREA : NAME->S_Dr9_Clng LENGTH->2 STARTBIT :34"}
GVL.IIVD.S_Dr9_Clng.v					:= NOT GVL.IIVD.S_TmOut_Kapi_Durum_3_0X238 AND NOT _FB_CanRx_Message_Unpack_238.S_Bit_35;
GVL.IIVD.S_Dr9_Clng.x					:= GVL.IIVD.S_Dr9_Clng.v AND _FB_CanRx_Message_Unpack_238.S_Bit_34;
GVL.IIVD.S_Dr9_Clng.e					:= _FB_CanRx_Message_Unpack_238.S_Bit_35 AND NOT _FB_CanRx_Message_Unpack_238.S_Bit_34 ;
GVL.IIVD.S_Dr9_Clng.na					:= _FB_CanRx_Message_Unpack_238.S_Bit_35 AND _FB_CanRx_Message_Unpack_238.S_Bit_34 ;
{endregion}
{region " SIGNAL AREA : NAME->S_Dr9_Op LENGTH->2 STARTBIT :36"}
GVL.IIVD.S_Dr9_Op.v						:= NOT GVL.IIVD.S_TmOut_Kapi_Durum_3_0X238 AND NOT _FB_CanRx_Message_Unpack_238.S_Bit_37;
GVL.IIVD.S_Dr9_Op.x						:= GVL.IIVD.S_Dr9_Op.v AND _FB_CanRx_Message_Unpack_238.S_Bit_36;
GVL.IIVD.S_Dr9_Op.e						:= _FB_CanRx_Message_Unpack_238.S_Bit_37 AND NOT _FB_CanRx_Message_Unpack_238.S_Bit_36 ;
GVL.IIVD.S_Dr9_Op.na					:= _FB_CanRx_Message_Unpack_238.S_Bit_37 AND _FB_CanRx_Message_Unpack_238.S_Bit_36 ;
{endregion}
{region " SIGNAL AREA : NAME->S_Dr9_Cl LENGTH->2 STARTBIT :38"}
GVL.IIVD.S_Dr9_Cl.v						:= NOT GVL.IIVD.S_TmOut_Kapi_Durum_3_0X238 AND NOT _FB_CanRx_Message_Unpack_238.S_Bit_39;
GVL.IIVD.S_Dr9_Cl.x						:= GVL.IIVD.S_Dr9_Cl.v AND _FB_CanRx_Message_Unpack_238.S_Bit_38;
GVL.IIVD.S_Dr9_Cl.e						:= _FB_CanRx_Message_Unpack_238.S_Bit_39 AND NOT _FB_CanRx_Message_Unpack_238.S_Bit_38 ;
GVL.IIVD.S_Dr9_Cl.na					:= _FB_CanRx_Message_Unpack_238.S_Bit_39 AND _FB_CanRx_Message_Unpack_238.S_Bit_38 ;
{endregion}
{region " SIGNAL AREA : NAME->S_Dr9_Obs LENGTH->2 STARTBIT :40"}
GVL.IIVD.S_Dr9_Obs.v					:= NOT GVL.IIVD.S_TmOut_Kapi_Durum_3_0X238 AND NOT _FB_CanRx_Message_Unpack_238.S_Bit_41;
GVL.IIVD.S_Dr9_Obs.x					:= GVL.IIVD.S_Dr9_Obs.v AND _FB_CanRx_Message_Unpack_238.S_Bit_40;
GVL.IIVD.S_Dr9_Obs.e					:= _FB_CanRx_Message_Unpack_238.S_Bit_41 AND NOT _FB_CanRx_Message_Unpack_238.S_Bit_40 ;
GVL.IIVD.S_Dr9_Obs.na					:= _FB_CanRx_Message_Unpack_238.S_Bit_41 AND _FB_CanRx_Message_Unpack_238.S_Bit_40 ;
{endregion}
{region " SIGNAL AREA : NAME->S_Dr9_Em_Swc LENGTH->2 STARTBIT :42"}
GVL.IIVD.S_Dr9_Em_Swc.v					:= NOT GVL.IIVD.S_TmOut_Kapi_Durum_3_0X238 AND NOT _FB_CanRx_Message_Unpack_238.S_Bit_43;
GVL.IIVD.S_Dr9_Em_Swc.x					:= GVL.IIVD.S_Dr9_Em_Swc.v AND _FB_CanRx_Message_Unpack_238.S_Bit_42;
GVL.IIVD.S_Dr9_Em_Swc.e					:= _FB_CanRx_Message_Unpack_238.S_Bit_43 AND NOT _FB_CanRx_Message_Unpack_238.S_Bit_42 ;
GVL.IIVD.S_Dr9_Em_Swc.na				:= _FB_CanRx_Message_Unpack_238.S_Bit_43 AND _FB_CanRx_Message_Unpack_238.S_Bit_42 ;
{endregion}
{endregion}

// PR1006_REV_002619_TIMTRO
{region " MESSAGE AREA :Sigorta_Kontrol_1- ID:260"}

_FB_CanRx_Message_Unpack_260 (		C_Enable	:= GVL.IIVD.S_CAN_Init,
     								Obj_CAN		:= ADR(GVL.IC.Obj_CAN0),
     								X_MsgID		:= 16#260,
     								Tm_MsgTmOut	:= TIME#5000MS,
     								S_Extended	:= 0,
     								S_ER_TmOut	=> GVL.IIVD.S_TmOut_Sigorta_Kontrol_1_0X260);

{region " SIGNAL AREA : NAME->X_Fus_0_D1 LENGTH->8 STARTBIT :0"}
Raw_X_Fus_0_D1							:= _FB_CanRx_Message_Unpack_260.X_Byte_7;
GVL.IIVD.X_Fus_0_D1.e					:= (Raw_X_Fus_0_D1 > 16#FD) AND (Raw_X_Fus_0_D1 < 16#FF);
GVL.IIVD.X_Fus_0_D1.na					:= (Raw_X_Fus_0_D1 = 16#FF);
GVL.IIVD.X_Fus_0_D1.RangeExcd			:= NOT (Raw_X_Fus_0_D1 >= 0) AND (Raw_X_Fus_0_D1 <= 254);
GVL.IIVD.X_Fus_0_D1.v					:= NOT( GVL.IIVD.S_TmOut_Sigorta_Kontrol_1_0X260 OR GVL.IIVD.X_Fus_0_D1.RangeExcd OR GVL.IIVD.X_Fus_0_D1.e OR GVL.IIVD.X_Fus_0_D1.na) ;
GVL.IIVD.X_Fus_0_D1.x					:= 
(*SELECT 1 : Is data valid ?*)				SEL(GVL.IIVD.X_Fus_0_D1.v,
(*DEFAULT value assigment*)					0,
(*Transmission is VALID*)					Raw_X_Fus_0_D1);


{endregion}
{region " SIGNAL AREA : NAME->X_Fus_0_D2 LENGTH->8 STARTBIT :8"}
Raw_X_Fus_0_D2							:= _FB_CanRx_Message_Unpack_260.X_Byte_6;
GVL.IIVD.X_Fus_0_D2.e					:= (Raw_X_Fus_0_D2 > 16#FD) AND (Raw_X_Fus_0_D2 < 16#FF);
GVL.IIVD.X_Fus_0_D2.na					:= (Raw_X_Fus_0_D2 = 16#FF);
GVL.IIVD.X_Fus_0_D2.RangeExcd			:= NOT (Raw_X_Fus_0_D2 >= 0) AND (Raw_X_Fus_0_D2 <= 254);
GVL.IIVD.X_Fus_0_D2.v					:= NOT( GVL.IIVD.S_TmOut_Sigorta_Kontrol_1_0X260 OR GVL.IIVD.X_Fus_0_D2.RangeExcd OR GVL.IIVD.X_Fus_0_D2.e OR GVL.IIVD.X_Fus_0_D2.na) ;
GVL.IIVD.X_Fus_0_D2.x					:= 
(*SELECT 1 : Is data valid ?*)				SEL(GVL.IIVD.X_Fus_0_D2.v,
(*DEFAULT value assigment*)					0,
(*Transmission is VALID*)					Raw_X_Fus_0_D2);


{endregion}
{region " SIGNAL AREA : NAME->X_Fus_0_D3 LENGTH->8 STARTBIT :16"}
Raw_X_Fus_0_D3							:= _FB_CanRx_Message_Unpack_260.X_Byte_5;
GVL.IIVD.X_Fus_0_D3.e					:= (Raw_X_Fus_0_D3 > 16#FD) AND (Raw_X_Fus_0_D3 < 16#FF);
GVL.IIVD.X_Fus_0_D3.na					:= (Raw_X_Fus_0_D3 = 16#FF);
GVL.IIVD.X_Fus_0_D3.RangeExcd			:= NOT (Raw_X_Fus_0_D3 >= 0) AND (Raw_X_Fus_0_D3 <= 254);
GVL.IIVD.X_Fus_0_D3.v					:= NOT( GVL.IIVD.S_TmOut_Sigorta_Kontrol_1_0X260 OR GVL.IIVD.X_Fus_0_D3.RangeExcd OR GVL.IIVD.X_Fus_0_D3.e OR GVL.IIVD.X_Fus_0_D3.na) ;
GVL.IIVD.X_Fus_0_D3.x					:= 
(*SELECT 1 : Is data valid ?*)				SEL(GVL.IIVD.X_Fus_0_D3.v,
(*DEFAULT value assigment*)					0,
(*Transmission is VALID*)					Raw_X_Fus_0_D3);

{endregion}
{region " SIGNAL AREA : NAME->X_Fus_0_D4 LENGTH->8 STARTBIT :24"}
Raw_X_Fus_0_D4							:= _FB_CanRx_Message_Unpack_260.X_Byte_4;
GVL.IIVD.X_Fus_0_D4.e					:= (Raw_X_Fus_0_D4 > 16#FD) AND (Raw_X_Fus_0_D4 < 16#FF);
GVL.IIVD.X_Fus_0_D4.na					:= (Raw_X_Fus_0_D4 = 16#FF);
GVL.IIVD.X_Fus_0_D4.RangeExcd			:= NOT (Raw_X_Fus_0_D4 >= 0) AND (Raw_X_Fus_0_D4 <= 254);
GVL.IIVD.X_Fus_0_D4.v					:= NOT( GVL.IIVD.S_TmOut_Sigorta_Kontrol_1_0X260 OR GVL.IIVD.X_Fus_0_D4.RangeExcd OR GVL.IIVD.X_Fus_0_D4.e OR GVL.IIVD.X_Fus_0_D4.na) ;
GVL.IIVD.X_Fus_0_D4.x					:= 
(*SELECT 1 : Is data valid ?*)				SEL(GVL.IIVD.X_Fus_0_D4.v,
(*DEFAULT value assigment*)					0,
(*Transmission is VALID*)					Raw_X_Fus_0_D4);


{endregion}
{region " SIGNAL AREA : NAME->X_Fus_0_D5 LENGTH->8 STARTBIT :32"}
Raw_X_Fus_0_D5							:= _FB_CanRx_Message_Unpack_260.X_Byte_3;
GVL.IIVD.X_Fus_0_D5.e					:= (Raw_X_Fus_0_D5 > 16#FD) AND (Raw_X_Fus_0_D5 < 16#FF);
GVL.IIVD.X_Fus_0_D5.na					:= (Raw_X_Fus_0_D5 = 16#FF);
GVL.IIVD.X_Fus_0_D5.RangeExcd			:= NOT (Raw_X_Fus_0_D5 >= 0) AND (Raw_X_Fus_0_D5 <= 254);
GVL.IIVD.X_Fus_0_D5.v					:= NOT( GVL.IIVD.S_TmOut_Sigorta_Kontrol_1_0X260 OR GVL.IIVD.X_Fus_0_D5.RangeExcd OR GVL.IIVD.X_Fus_0_D5.e OR GVL.IIVD.X_Fus_0_D5.na) ;
GVL.IIVD.X_Fus_0_D5.x					:= 
(*SELECT 1 : Is data valid ?*)				SEL(GVL.IIVD.X_Fus_0_D5.v,
(*DEFAULT value assigment*)					0,
(*Transmission is VALID*)					Raw_X_Fus_0_D5);


{endregion}
{region " SIGNAL AREA : NAME->X_Fus_0_D6 LENGTH->8 STARTBIT :40"}
Raw_X_Fus_0_D6							:= _FB_CanRx_Message_Unpack_260.X_Byte_2;
GVL.IIVD.X_Fus_0_D6.e					:= (Raw_X_Fus_0_D6 > 16#FD) AND (Raw_X_Fus_0_D6 < 16#FF);
GVL.IIVD.X_Fus_0_D6.na					:= (Raw_X_Fus_0_D6 = 16#FF);
GVL.IIVD.X_Fus_0_D6.RangeExcd			:= NOT (Raw_X_Fus_0_D6 >= 0) AND (Raw_X_Fus_0_D6 <= 254);
GVL.IIVD.X_Fus_0_D6.v					:= NOT( GVL.IIVD.S_TmOut_Sigorta_Kontrol_1_0X260 OR GVL.IIVD.X_Fus_0_D6.RangeExcd OR GVL.IIVD.X_Fus_0_D6.e OR GVL.IIVD.X_Fus_0_D6.na) ;
GVL.IIVD.X_Fus_0_D6.x					:= 
(*SELECT 1 : Is data valid ?*)				SEL(GVL.IIVD.X_Fus_0_D6.v,
(*DEFAULT value assigment*)					0,
(*Transmission is VALID*)					Raw_X_Fus_0_D6);


{endregion}
{region " SIGNAL AREA : NAME->X_Fus_0_D7 LENGTH->8 STARTBIT :48"}
Raw_X_Fus_0_D7							:= _FB_CanRx_Message_Unpack_260.X_Byte_1;
GVL.IIVD.X_Fus_0_D7.e					:= (Raw_X_Fus_0_D7 > 16#FD) AND (Raw_X_Fus_0_D7 < 16#FF);
GVL.IIVD.X_Fus_0_D7.na					:= (Raw_X_Fus_0_D7 = 16#FF);
GVL.IIVD.X_Fus_0_D7.RangeExcd			:= NOT (Raw_X_Fus_0_D7 >= 0) AND (Raw_X_Fus_0_D7 <= 254);
GVL.IIVD.X_Fus_0_D7.v					:= NOT( GVL.IIVD.S_TmOut_Sigorta_Kontrol_1_0X260 OR GVL.IIVD.X_Fus_0_D7.RangeExcd OR GVL.IIVD.X_Fus_0_D7.e OR GVL.IIVD.X_Fus_0_D7.na) ;
GVL.IIVD.X_Fus_0_D7.x					:= 
(*SELECT 1 : Is data valid ?*)				SEL(GVL.IIVD.X_Fus_0_D7.v,
(*DEFAULT value assigment*)					0,
(*Transmission is VALID*)					Raw_X_Fus_0_D7);


{endregion}
{region " SIGNAL AREA : NAME->S_Fus_0_5 LENGTH->8 STARTBIT :56"}
Raw_X_Fus_0_D8							:= _FB_CanRx_Message_Unpack_260.X_Byte_0;
GVL.IIVD.X_Fus_0_D8.e					:= (Raw_X_Fus_0_D8 > 16#FD) AND (Raw_X_Fus_0_D8 < 16#FF);
GVL.IIVD.X_Fus_0_D8.na					:= (Raw_X_Fus_0_D8 = 16#FF);
GVL.IIVD.X_Fus_0_D8.RangeExcd			:= NOT (Raw_X_Fus_0_D8 >= 0) AND (Raw_X_Fus_0_D8 <= 254);
GVL.IIVD.X_Fus_0_D8.v					:= NOT( GVL.IIVD.S_TmOut_Sigorta_Kontrol_1_0X260 OR GVL.IIVD.X_Fus_0_D8.RangeExcd OR GVL.IIVD.X_Fus_0_D8.e OR GVL.IIVD.X_Fus_0_D8.na) ;
GVL.IIVD.X_Fus_0_D8.x					:= 
(*SELECT 1 : Is data valid ?*)				SEL(GVL.IIVD.X_Fus_0_D8.v,
(*DEFAULT value assigment*)					0,
(*Transmission is VALID*)					Raw_X_Fus_0_D8);

//PR1006_REV_002685_TIMTRO
GVL.EF.S_Fus_0_01						:= GVL.IIVD.X_Fus_0_D1.v AND _FB_CanRx_Message_Unpack_260.S_Bit_6;
GVL.EF.S_Fus_0_02						:= GVL.IIVD.X_Fus_0_D1.v AND _FB_CanRx_Message_Unpack_260.S_Bit_4;
GVL.EF.S_Fus_0_03						:= GVL.IIVD.X_Fus_0_D1.v AND _FB_CanRx_Message_Unpack_260.S_Bit_2;
GVL.EF.S_Fus_0_04						:= GVL.IIVD.X_Fus_0_D1.v AND _FB_CanRx_Message_Unpack_260.S_Bit_0;	  
GVL.EF.S_Fus_0_05						:= GVL.IIVD.X_Fus_0_D2.v AND _FB_CanRx_Message_Unpack_260.S_Bit_14;
GVL.EF.S_Fus_0_06						:= GVL.IIVD.X_Fus_0_D2.v AND _FB_CanRx_Message_Unpack_260.S_Bit_12;
GVL.EF.S_Fus_0_07						:= GVL.IIVD.X_Fus_0_D2.v AND _FB_CanRx_Message_Unpack_260.S_Bit_10;
GVL.EF.S_Fus_0_08						:= GVL.IIVD.X_Fus_0_D2.v AND _FB_CanRx_Message_Unpack_260.S_Bit_8;					
GVL.EF.S_Fus_0_09						:= GVL.IIVD.X_Fus_0_D3.v AND _FB_CanRx_Message_Unpack_260.S_Bit_22;
GVL.EF.S_Fus_0_10						:= GVL.IIVD.X_Fus_0_D3.v AND _FB_CanRx_Message_Unpack_260.S_Bit_20;
GVL.EF.S_Fus_0_11						:= GVL.IIVD.X_Fus_0_D3.v AND _FB_CanRx_Message_Unpack_260.S_Bit_18;
GVL.EF.S_Fus_0_12						:= GVL.IIVD.X_Fus_0_D3.v AND _FB_CanRx_Message_Unpack_260.S_Bit_16;							  
GVL.EF.S_Fus_0_13						:= GVL.IIVD.X_Fus_0_D4.v AND _FB_CanRx_Message_Unpack_260.S_Bit_30;
GVL.EF.S_Fus_0_14						:= GVL.IIVD.X_Fus_0_D4.v AND _FB_CanRx_Message_Unpack_260.S_Bit_28;
GVL.EF.S_Fus_0_15						:= GVL.IIVD.X_Fus_0_D4.v AND _FB_CanRx_Message_Unpack_260.S_Bit_26;
GVL.EF.S_Fus_0_16						:= GVL.IIVD.X_Fus_0_D4.v AND _FB_CanRx_Message_Unpack_260.S_Bit_24;										
GVL.EF.S_Fus_0_17						:= GVL.IIVD.X_Fus_0_D5.v AND _FB_CanRx_Message_Unpack_260.S_Bit_38;
GVL.EF.S_Fus_0_18						:= GVL.IIVD.X_Fus_0_D5.v AND _FB_CanRx_Message_Unpack_260.S_Bit_36;
GVL.EF.S_Fus_0_19						:= GVL.IIVD.X_Fus_0_D5.v AND _FB_CanRx_Message_Unpack_260.S_Bit_34;
GVL.EF.S_Fus_0_20						:= GVL.IIVD.X_Fus_0_D5.v AND _FB_CanRx_Message_Unpack_260.S_Bit_32;		  
GVL.EF.S_Fus_0_21						:= GVL.IIVD.X_Fus_0_D6.v AND _FB_CanRx_Message_Unpack_260.S_Bit_46;
GVL.EF.S_Fus_0_22						:= GVL.IIVD.X_Fus_0_D6.v AND _FB_CanRx_Message_Unpack_260.S_Bit_44;
GVL.EF.S_Fus_0_23						:= GVL.IIVD.X_Fus_0_D6.v AND _FB_CanRx_Message_Unpack_260.S_Bit_42;
GVL.EF.S_Fus_0_24						:= GVL.IIVD.X_Fus_0_D6.v AND _FB_CanRx_Message_Unpack_260.S_Bit_40;		  
GVL.EF.S_Fus_0_25						:= GVL.IIVD.X_Fus_0_D7.v AND _FB_CanRx_Message_Unpack_260.S_Bit_54;
GVL.EF.S_Fus_0_26						:= GVL.IIVD.X_Fus_0_D7.v AND _FB_CanRx_Message_Unpack_260.S_Bit_52;
GVL.EF.S_Fus_0_27						:= GVL.IIVD.X_Fus_0_D7.v AND _FB_CanRx_Message_Unpack_260.S_Bit_50;
GVL.EF.S_Fus_0_28						:= GVL.IIVD.X_Fus_0_D7.v AND _FB_CanRx_Message_Unpack_260.S_Bit_48;											  
GVL.EF.S_Fus_0_29						:= GVL.IIVD.X_Fus_0_D8.v AND _FB_CanRx_Message_Unpack_260.S_Bit_62;
GVL.EF.S_Fus_0_30						:= GVL.IIVD.X_Fus_0_D8.v AND _FB_CanRx_Message_Unpack_260.S_Bit_60;
{endregion}
{endregion}

// PR1006_REV_002619_TIMTRO
{region " MESSAGE AREA :Sigorta_Kontrol_2- ID:261"}
_FB_CanRx_Message_Unpack_261 (		C_Enable	:= GVL.IIVD.S_CAN_Init,
     								Obj_CAN		:= ADR(GVL.IC.Obj_CAN0),
     								X_MsgID		:= 16#261,
     								Tm_MsgTmOut	:= TIME#2500MS,
     								S_Extended	:= 0,
     								S_ER_TmOut	=> GVL.IIVD.S_TmOut_Sigorta_Kontrol_2_0X261);

{region " SIGNAL AREA : NAME->X_Fus_1_D1 LENGTH->8 STARTBIT :0"}
Raw_X_Fus_1_D1							:= _FB_CanRx_Message_Unpack_261.X_Byte_7;
GVL.IIVD.X_Fus_1_D1.e					:= (Raw_X_Fus_1_D1 > 16#FD) AND (Raw_X_Fus_1_D1 < 16#FF);
GVL.IIVD.X_Fus_1_D1.na					:= (Raw_X_Fus_1_D1 = 16#FF);
GVL.IIVD.X_Fus_1_D1.RangeExcd			:= NOT (Raw_X_Fus_0_D1 >= 0) AND (Raw_X_Fus_1_D1 <= 254);
GVL.IIVD.X_Fus_1_D1.v					:= NOT( GVL.IIVD.S_TmOut_Sigorta_Kontrol_2_0X261 OR GVL.IIVD.X_Fus_1_D1.RangeExcd OR GVL.IIVD.X_Fus_1_D1.e OR GVL.IIVD.X_Fus_1_D1.na) ;
GVL.IIVD.X_Fus_1_D1.x					:= 
(*SELECT 1 : Is data valid ?*)				SEL(GVL.IIVD.X_Fus_1_D1.v,
(*DEFAULT value assigment*)					0,
(*Transmission is VALID*)					Raw_X_Fus_1_D1);

{endregion}
{region " SIGNAL AREA : NAME->X_Fus_1_D2 LENGTH->8 STARTBIT :8"}
Raw_X_Fus_1_D2							:= _FB_CanRx_Message_Unpack_261.X_Byte_6;
GVL.IIVD.X_Fus_1_D2.e					:= (Raw_X_Fus_1_D2 > 16#FD) AND (Raw_X_Fus_1_D2 < 16#FF);
GVL.IIVD.X_Fus_1_D2.na					:= (Raw_X_Fus_1_D2 = 16#FF);
GVL.IIVD.X_Fus_1_D2.RangeExcd			:= NOT (Raw_X_Fus_0_D1 >= 0) AND (Raw_X_Fus_1_D2 <= 254);
GVL.IIVD.X_Fus_1_D2.v					:= NOT( GVL.IIVD.S_TmOut_Sigorta_Kontrol_2_0X261 OR GVL.IIVD.X_Fus_1_D2.RangeExcd OR GVL.IIVD.X_Fus_1_D2.e OR GVL.IIVD.X_Fus_1_D2.na) ;
GVL.IIVD.X_Fus_1_D2.x					:= 
(*SELECT 1 : Is data valid ?*)				SEL(GVL.IIVD.X_Fus_1_D2.v,
(*DEFAULT value assigment*)					0,
(*Transmission is VALID*)					Raw_X_Fus_1_D2);

{endregion}
{region " SIGNAL AREA : NAME->X_Fus_1_D3 LENGTH->8 STARTBIT :16"}
Raw_X_Fus_1_D3							:= _FB_CanRx_Message_Unpack_261.X_Byte_5;
GVL.IIVD.X_Fus_1_D3.e					:= (Raw_X_Fus_1_D3 > 16#FD) AND (Raw_X_Fus_1_D3 < 16#FF);
GVL.IIVD.X_Fus_1_D3.na					:= (Raw_X_Fus_1_D3 = 16#FF);
GVL.IIVD.X_Fus_1_D3.RangeExcd			:= NOT (Raw_X_Fus_0_D1 >= 0) AND (Raw_X_Fus_1_D3 <= 254);
GVL.IIVD.X_Fus_1_D3.v					:= NOT( GVL.IIVD.S_TmOut_Sigorta_Kontrol_2_0X261 OR GVL.IIVD.X_Fus_1_D3.RangeExcd OR GVL.IIVD.X_Fus_1_D3.e OR GVL.IIVD.X_Fus_1_D3.na) ;
GVL.IIVD.X_Fus_1_D3.x					:= 
(*SELECT 1 : Is data valid ?*)				SEL(GVL.IIVD.X_Fus_1_D3.v,
(*DEFAULT value assigment*)					0,
(*Transmission is VALID*)					Raw_X_Fus_1_D3);

{endregion}
{region " SIGNAL AREA : NAME->X_Fus_1_D4 LENGTH->8 STARTBIT :24"}
Raw_X_Fus_1_D4							:= _FB_CanRx_Message_Unpack_261.X_Byte_4;
GVL.IIVD.X_Fus_1_D4.e					:= (Raw_X_Fus_1_D4 > 16#FD) AND (Raw_X_Fus_1_D4 < 16#FF);
GVL.IIVD.X_Fus_1_D4.na					:= (Raw_X_Fus_1_D4 = 16#FF);
GVL.IIVD.X_Fus_1_D4.RangeExcd			:= NOT (Raw_X_Fus_0_D1 >= 0) AND (Raw_X_Fus_1_D4 <= 254);
GVL.IIVD.X_Fus_1_D4.v					:= NOT( GVL.IIVD.S_TmOut_Sigorta_Kontrol_2_0X261 OR GVL.IIVD.X_Fus_1_D4.RangeExcd OR GVL.IIVD.X_Fus_1_D4.e OR GVL.IIVD.X_Fus_1_D4.na) ;
GVL.IIVD.X_Fus_1_D4.x					:= 
(*SELECT 1 : Is data valid ?*)				SEL(GVL.IIVD.X_Fus_1_D4.v,
(*DEFAULT value assigment*)					0,
(*Transmission is VALID*)					Raw_X_Fus_1_D4);

{endregion}
{region " SIGNAL AREA : NAME->X_Fus_1_D5 LENGTH->8 STARTBIT :32"}
Raw_X_Fus_1_D5							:= _FB_CanRx_Message_Unpack_261.X_Byte_3;
GVL.IIVD.X_Fus_1_D5.e					:= (Raw_X_Fus_1_D5 > 16#FD) AND (Raw_X_Fus_1_D5 < 16#FF);
GVL.IIVD.X_Fus_1_D5.na					:= (Raw_X_Fus_1_D5 = 16#FF);
GVL.IIVD.X_Fus_1_D5.RangeExcd			:= NOT (Raw_X_Fus_0_D1 >= 0) AND (Raw_X_Fus_1_D5 <= 254);
GVL.IIVD.X_Fus_1_D5.v					:= NOT( GVL.IIVD.S_TmOut_Sigorta_Kontrol_2_0X261 OR GVL.IIVD.X_Fus_1_D5.RangeExcd OR GVL.IIVD.X_Fus_1_D5.e OR GVL.IIVD.X_Fus_1_D5.na) ;
GVL.IIVD.X_Fus_1_D5.x					:= 
(*SELECT 1 : Is data valid ?*)				SEL(GVL.IIVD.X_Fus_1_D5.v,
(*DEFAULT value assigment*)					0,
(*Transmission is VALID*)					Raw_X_Fus_1_D5);

{endregion}
{region " SIGNAL AREA : NAME->X_Fus_1_D6 LENGTH->8 STARTBIT :40"}
Raw_X_Fus_1_D6							:= _FB_CanRx_Message_Unpack_261.X_Byte_2;
GVL.IIVD.X_Fus_1_D6.e					:= (Raw_X_Fus_1_D6 > 16#FD) AND (Raw_X_Fus_1_D6 < 16#FF);
GVL.IIVD.X_Fus_1_D6.na					:= (Raw_X_Fus_1_D6 = 16#FF);
GVL.IIVD.X_Fus_1_D6.RangeExcd			:= NOT (Raw_X_Fus_0_D1 >= 0) AND (Raw_X_Fus_1_D6 <= 254);
GVL.IIVD.X_Fus_1_D6.v					:= NOT( GVL.IIVD.S_TmOut_Sigorta_Kontrol_2_0X261 OR GVL.IIVD.X_Fus_1_D6.RangeExcd OR GVL.IIVD.X_Fus_1_D6.e OR GVL.IIVD.X_Fus_1_D6.na) ;
GVL.IIVD.X_Fus_1_D6.x					:= 
(*SELECT 1 : Is data valid ?*)				SEL(GVL.IIVD.X_Fus_1_D6.v,
(*DEFAULT value assigment*)					0,
(*Transmission is VALID*)					Raw_X_Fus_1_D6);

{endregion}
{region " SIGNAL AREA : NAME->X_Fus_1_D7 LENGTH->8 STARTBIT :48"}
Raw_X_Fus_1_D7							:= _FB_CanRx_Message_Unpack_261.X_Byte_1;
GVL.IIVD.X_Fus_1_D7.e					:= (Raw_X_Fus_1_D7 > 16#FD) AND (Raw_X_Fus_1_D7 < 16#FF);
GVL.IIVD.X_Fus_1_D7.na					:= (Raw_X_Fus_1_D7 = 16#FF);
GVL.IIVD.X_Fus_1_D7.RangeExcd			:= NOT (Raw_X_Fus_0_D1 >= 0) AND (Raw_X_Fus_1_D7 <= 254);
GVL.IIVD.X_Fus_1_D7.v					:= NOT( GVL.IIVD.S_TmOut_Sigorta_Kontrol_2_0X261 OR GVL.IIVD.X_Fus_1_D7.RangeExcd OR GVL.IIVD.X_Fus_1_D7.e OR GVL.IIVD.X_Fus_1_D7.na) ;
GVL.IIVD.X_Fus_1_D7.x					:= 
(*SELECT 1 : Is data valid ?*)				SEL(GVL.IIVD.X_Fus_1_D7.v,
(*DEFAULT value assigment*)					0,
(*Transmission is VALID*)					Raw_X_Fus_1_D7);

{endregion}
{region " SIGNAL AREA : NAME->X_Fus_1_D8 LENGTH->8 STARTBIT :56"}
Raw_X_Fus_1_D8							:= _FB_CanRx_Message_Unpack_261.X_Byte_0;
GVL.IIVD.X_Fus_1_D8.e					:= (Raw_X_Fus_1_D8 > 16#FD) AND (Raw_X_Fus_1_D8 < 16#FF);
GVL.IIVD.X_Fus_1_D8.na					:= (Raw_X_Fus_1_D8 = 16#FF);
GVL.IIVD.X_Fus_1_D8.RangeExcd			:= NOT (Raw_X_Fus_0_D1 >= 0) AND (Raw_X_Fus_1_D8 <= 254);
GVL.IIVD.X_Fus_1_D8.v					:= NOT( GVL.IIVD.S_TmOut_Sigorta_Kontrol_2_0X261 OR GVL.IIVD.X_Fus_1_D8.RangeExcd OR GVL.IIVD.X_Fus_1_D8.e OR GVL.IIVD.X_Fus_1_D8.na) ;
GVL.IIVD.X_Fus_1_D8.x					:= 
(*SELECT 1 : Is data valid ?*)				SEL(GVL.IIVD.X_Fus_1_D8.v,
(*DEFAULT value assigment*)					0,
(*Transmission is VALID*)					Raw_X_Fus_1_D8);

